# B&R Automation Studio project TD52 (part 74)

#### LX2.c
```c
/********************************************************************
 * COPYRIGHT -- Bernecker + Rainer Industrie-Elektronik Ges.m.b.H.
 ********************************************************************
 * Program: LX2
 * File: LX2.c
 * Author: 212566120
 * Created: Wed Apr 11 13:34:17 2018
 ********************************************************************
 * Implementation of program LX2
 ********************************************************************
 * Generated with B&R Automation Studio Target for Simulink V4.2
 * (ERT based)
 ********************************************************************/
#include "LX2.h"
#include "LX2_private.h"

/*  Defines */
#define LX2_POS_ZCSIG                  ((uint8_T)1U)
#define LX2_UNINITIALIZED_ZCSIG        ((uint8_T)3U)

/*  Data Types */

/**************************** GLOBAL DATA *************************************/
/*  Definitions */

/* Block signals (auto storage) */
struct BlockIO_LX2 LX2_B;

/* Block states (auto storage) */
struct D_Work_LX2 LX2_DWork;

/* Previous zero-crossings (trigger) states */
struct PrevZCSigStates_LX2 LX2_PrevZCSigState;

/* External inputs (root inport signals with auto storage) */
ExternalInputs_LX2 LX2_U;

/* External outputs (root outports fed by signals with auto storage) */
ExternalOutputs_LX2 LX2_Y;

/* Real-time model */
RT_MODEL_LX2 LX2_M_;
RT_MODEL_LX2 *const LX2_M = &LX2_M_;

/*  Declarations  */

/* Forward declaration for local functions */
static void LX2_my_split(real32_T x, real32_T *b_y1, real32_T *y2, struct fLX2* inst);
static void LX2_my_detect(real32_T x, real32_T *x1, real32_T *x2, struct fLX2* inst);
static real32_T LX2_my_split_i(real32_T x, struct fLX2* inst);
static void LX2_my_find(const real32_T V[11], real_T LowerLimit, real32_T
  UpperLimit, real_T p[11], struct fLX2* inst);
static void LX2_my_find_e(const real32_T V[11], real_T LowerLimit, real32_T
  UpperLimit, real_T p[11], struct fLX2* inst);
static void LX2_my_find_ex(const real32_T V[11], real32_T LowerLimit, real32_T
  UpperLimit, real_T p[11], struct fLX2* inst);
static void LX2_my_find_exl(const real32_T V[11], real32_T LowerLimit, real32_T
  UpperLimit, real_T p[11], struct fLX2* inst);
static void LX2_my_find_exlq(const real32_T V[11], real32_T LowerLimit, real_T
  UpperLimit, real_T p[11], struct fLX2* inst);
static void LX2_my_find_exlqw(const real32_T V[11], real32_T LowerLimit, real_T
  UpperLimit, real_T p[11], struct fLX2* inst);
static void LX2_my_find_exlqwy(const real32_T V[11], real_T p[11], struct fLX2* inst);
static real32_T LX2_sum(const real32_T x[11], struct fLX2* inst);
static void LX2_my_smoothing(const real32_T Pl[2], real32_T Pm[2], const
  real32_T Pr[2], real32_T slope_max, struct fLX2* inst);
static void LX2_interp1(const real32_T varargin_1[3], const real32_T varargin_2
  [3], const real32_T varargin_3[11], real32_T yi[11], struct fLX2* inst);
static void LX2_interp1_o(const real32_T varargin_1[4], const real32_T
  varargin_2[4], const real32_T varargin_3[11], real32_T yi[11], struct fLX2* inst);
static void LX2_interp1_o5pn4ly1(const real32_T varargin_1[11], const real32_T
  varargin_2[11], const real32_T varargin_3[11], real32_T yi[11], struct fLX2* inst);
static void LX2_interp1_o5(const real32_T varargin_1[5], const real32_T
  varargin_2[5], const real32_T varargin_3[11], real32_T yi[11], struct fLX2* inst);
static void LX2_interp1_o5p(const real32_T varargin_1[6], const real32_T
  varargin_2[6], const real32_T varargin_3[11], real32_T yi[11], struct fLX2* inst);
static void LX2_interp1_o5pn(const real32_T varargin_1[7], const real32_T
  varargin_2[7], const real32_T varargin_3[11], real32_T yi[11], struct fLX2* inst);
static real32_T LX2_interp1_o5pn4ly1e(const real32_T varargin_1[2], const
  real32_T varargin_2[2], real32_T varargin_3, struct fLX2* inst);
static void LX2_interp1_o5pn4(const real32_T varargin_1[8], const real32_T
  varargin_2[8], const real32_T varargin_3[11], real32_T yi[11], struct fLX2* inst);
static void LX2_interp1_o5pn4l(const real32_T varargin_1[9], const real32_T
  varargin_2[9], const real32_T varargin_3[11], real32_T yi[11], struct fLX2* inst);
static void LX2_interp1_o5pn4ly(const real32_T varargin_1[10], const real32_T
  varargin_2[10], const real32_T varargin_3[11], real32_T yi[11], struct fLX2* inst);
static void LX2_rdivide(const real32_T x[4], real_T y, real32_T z[4], struct fLX2* inst);

/* Forward declaration for local functions */
static void LX2_my_BPOC_enable_h(const real32_T splitfactor[4], boolean_T
  bLX2_enable, const real32_T rThreshold_save2map[2], boolean_T
  bExt_BPOC_learning_Stop, boolean_T bBPOC_enable[4], boolean_T
  bSave_BPOC_enable[4], struct fLX2* inst);
static void LX2_my_BPOC_enable(const real32_T splitfactor[4], boolean_T
  bLX2_enable, const real32_T rThreshold_save2map[2], boolean_T
  bExt_BPOC_learning_Stop, boolean_T bBPOC_enable[4], boolean_T
  bSave_BPOC_enable[4], struct fLX2* inst);
static void LX2_my_gasmixing(uint16_T iIdx_Gtyp_Dem, real32_T rGT_QualMix_1_2,
  real32_T rGT_RatioMix, boolean_T bLX2_enable, const real32_T
  rThreshold_save2map[2], boolean_T bExt_BPOC_learning_Stop, real32_T
  splitfactor_Gas[4], boolean_T bBPOC_enable[4], boolean_T bSave_BPOC_enable[4], struct fLX2* inst);

/***************************** FILE SCOPE DATA ********************************/

/*************************** FUNCTIONS ****************************************/

/* Lookup Binary Search Utility BINARYSEARCH_real32_T */
void BINARYSEARCH_real32_T(uint32_T *piLeft, uint32_T *piRght, real32_T u, const
  real32_T *pData, uint32_T iHi, struct fLX2* inst)
{
  /* Find the location of current input value in the data table. */
  *piLeft = 0U;
  *piRght = iHi;
  if (u <= pData[0] ) {
    /* Less than or equal to the smallest point in the table. */
    *piRght = 0U;
  } else if (u >= pData[iHi] ) {
    /* Greater than or equal to the largest point in the table. */
    *piLeft = iHi;
  } else {
    uint32_T i;

    /* Do a binary search. */
    while (( *piRght - *piLeft ) > 1U ) {
      /* Get the average of the left and right indices using to Floor rounding. */
      i = (*piLeft + *piRght) >> 1;

      /* Move either the right index or the left index so that */
      /*  LeftDataPoint <= CurrentValue < RightDataPoint */
      if (u < pData[i] ) {
        *piRght = i;
      } else {
        *piLeft = i;
      }
    }
  }
}

/* Lookup Utility LookUp_real32_T_real32_T */
void LookUp_real32_T_real32_T(real32_T *pY, const real32_T *pYData, real32_T u,
  const real32_T *pUData, uint32_T iHi, struct fLX2* inst)
{
  uint32_T iLeft;
  uint32_T iRght;
  BINARYSEARCH_real32_T( &(iLeft), &(iRght), u, pUData, iHi, inst);

  {
    real32_T lambda;
    if (pUData[iRght] > pUData[iLeft] ) {
      real32_T num;
      real32_T den;
      den = pUData[iRght];
      den = den - pUData[iLeft];
      num = u;
      num = num - pUData[iLeft];
      lambda = num / den;
    } else {
      lambda = 0.0F;
    }

    {
      real32_T yLeftCast;
      real32_T yRghtCast;
      yLeftCast = pYData[iLeft];
      yRghtCast = pYData[iRght];
      yLeftCast += lambda * ( yRghtCast - yLeftCast );
      (*pY) = yLeftCast;
    }
  }
}

real32_T rt_roundf(real32_T u, struct fLX2* inst)
{
  real32_T y;
  if ((real32_T)fabs(u) < 8.388608E+6F) {
    if (u >= 0.5F) {
      y = (real32_T)floor(u + 0.5F);
    } else if (u > -0.5F) {
      y = 0.0F;
    } else {
      y = (real32_T)ceil(u - 0.5F);
    }
  } else {
    y = u;
  }

  return y;
}

/* Function for MATLAB Function: '<S10>/Boost Pressure Offset Curve' */
static void LX2_my_split(real32_T x, real32_T *b_y1, real32_T *y2, struct fLX2* inst)
{
  real32_T t;

  /*  End od 'my_detect-function' */
  /*  ---------------------------------------------------------------------------------- */
  /* % my_split function */
  /* ************************************************************************** */
  /*  divides new measurement value up to neighborhood node points via leverage function */
  /*  */
  /*  Input:    x   ... Engine Power [%] */
  /*  Output:   y1  ... weighting of node left from x [-] */
  /*                  y2  ... weighting of node right from x [-] */
  /* ************************************************************************** */
  t = rt_roundf(x / 10.0F, inst) * 10.0F;

  /*  temporary var for decision and find neighborhood point */
  if (x < t) {
    /*  slope between the two neighboring points is positive */
    t -= x;
    *y2 = 1.0F - t / 10.0F;

    /*  weighting of node right from x */
    *b_y1 = 1.0F - (1.0F - t / 10.0F);

    /*  weighting of node left from x */
  } else if (x > t) {
    /*  slope between the two neighboring points is negative */
    t = x - t;
    *b_y1 = 1.0F - t / 10.0F;

    /*  weighting of node left from x */
    *y2 = 1.0F - (1.0F - t / 10.0F);

    /*  weighting of node right from x */
  } else if ((x == t) && (x != 100.0F)) {
    /*  x is exactly on node point; weighting factor is 1 */
    *b_y1 = 1.0F;
    *y2 = 0.0F;
  } else {
    /*  x is 100 */
    *b_y1 = 0.0F;
    *y2 = 1.0F;
  }
}

/* Function for MATLAB Function: '<S10>/Boost Pressure Offset Curve' */
static void LX2_my_detect(real32_T x, real32_T *x1, real32_T *x2, struct fLX2* inst)
{
  /*  End od 'BPOC.m' */
  /*  ---------------------------------------------------------------------------------- */
  /* % my_detect function */
  /* ************************************************************************** */
  /*  returns indices of affected node points due to new measurement value */
  /*  */
  /*  Input:    x   ... Engine Power [%] */
  /*  Output:   x1  ... index of left neighbouring node point [-] */
  /*                  x2  ... index of right neighbouring node point [-] */
  /* ************************************************************************** */
  if (!(x - (real32_T)floor(x / 2.0F) * 2.0F != 0.0F)) {
    /*  if x is exaclty on node -> manipulate x value with a super small value so that it is not lying on node anymore ;-) */
    x += 0.001F;
  }

  if (x <= 0.0F) {
    /*  input is limited to positive values  */
    *x1 = 1.0F;
    *x2 = 2.0F;
  } else if (x >= 100.0F) {
    /*  input is limited to values smaller than 100 (full load) */
    *x1 = 10.0F;
    *x2 = 11.0F;
  } else {
    *x1 = (real32_T)ceil(x / 10.0F);
    *x2 = *x1 + 1.0F;
  }
}

/* Function for MATLAB Function: '<S10>/Boost Pressure Offset Curve' */
static real32_T LX2_my_split_i(real32_T x, struct fLX2* inst)
{
  real32_T b_y1;
  real32_T t;

  /*  End od 'my_detect-function' */
  /*  ---------------------------------------------------------------------------------- */
  /* % my_split function */
  /* ************************************************************************** */
  /*  divides new measurement value up to neighborhood node points via leverage function */
  /*  */
  /*  Input:    x   ... Engine Power [%] */
  /*  Output:   y1  ... weighting of node left from x [-] */
  /*                  y2  ... weighting of node right from x [-] */
  /* ************************************************************************** */
  t = rt_roundf(x / 10.0F, inst) * 10.0F;

  /*  temporary var for decision and find neighborhood point */
  if (x < t) {
    /*  slope between the two neighboring points is positive */
    /*  weighting of node right from x */
    b_y1 = 1.0F - (1.0F - (t - x) / 10.0F);

    /*  weighting of node left from x */
  } else if (x > t) {
    /*  slope between the two neighboring points is negative */
    b_y1 = 1.0F - (x - t) / 10.0F;

    /*  weighting of node left from x */
    /*  weighting of node right from x */
  } else if ((x == t) && (x != 100.0F)) {
    /*  x is exactly on node point; weighting factor is 1 */
    b_y1 = 1.0F;
  } else {
    /*  x is 100 */
    b_y1 = 0.0F;
  }

  return b_y1;
}

/* Function for MATLAB Function: '<S10>/Boost Pressure Offset Curve' */
static void LX2_my_find(const real32_T V[11], real_T LowerLimit, real32_T
  UpperLimit, real_T p[11], struct fLX2* inst)
{
  real32_T i;
  int32_T b_i;
  int32_T b;
  int32_T i_0;

  /*  end of 'my_smoothing-function' */
  /* ---------------------------------------------------------------------------------- */
  /* % my_find */
  /* ************************************************************************** */
  /*  returns indices of already measured points depending on 'mode' and 'Limits' */
  /*  */
  /*  Input:    V                   ... binary map (vector, 11 elements, boolean) */
  /*                LowerLimit   ... lower search boundary (scalar) */
  /*                UpperLimit   ... upper search boundary (scalar) */
  /*                mode            ... 'first' -> returns first 2 indices */
  /*                                      ... 'last' -> returns last 2 indices */
  /*                                      ... 'all' -> returns all found indices */
  /*  */
  /*  Output: Pm	...	middle point of triangle  (vector, 2 elements, Pm(1)->[%], Pm(2)->[mbar]) */
  /* ************************************************************************** */
  for (i_0 = 0; i_0 < 11; i_0++) {
    p[i_0] = 0.0;
  }

  /*  fixed allocated vector for saving indices */
  /*  -> function will return indices of first two elements which were found */
  /*  -> always write 2 values to p - no need for more, thats why 2=hard coded */
  i_0 = 0;
  b = (int32_T)((1.0F - (real32_T)LowerLimit) + UpperLimit);
  for (b_i = 0; b_i < b; b_i++) {
    i = (real32_T)LowerLimit + (real32_T)b_i;
    if ((V[(int32_T)i - 1] != 0.0F) && (i_0 < 2)) {
      p[i_0] = i;
      i_0++;
    }
  }

  /*  -> function will return indices of last two elements which were found        */
  /*  -> always write 2 values to p - no need for more, thats why 2=hard coded   */
  /*  end 'if-function' */
  /*  end of 'my_find-function'  */
  /* ---------------------------------------------------------------------------------- */
}

/* Function for MATLAB Function: '<S10>/Boost Pressure Offset Curve' */
static void LX2_my_find_e(const real32_T V[11], real_T LowerLimit, real32_T
  UpperLimit, real_T p[11], struct fLX2* inst)
{
  real32_T i;
  int32_T b_i;
  int32_T b;
  int32_T i_0;

  /*  end of 'my_smoothing-function' */
  /* ---------------------------------------------------------------------------------- */
  /* % my_find */
  /* ************************************************************************** */
  /*  returns indices of already measured points depending on 'mode' and 'Limits' */
  /*  */
  /*  Input:    V                   ... binary map (vector, 11 elements, boolean) */
  /*                LowerLimit   ... lower search boundary (scalar) */
  /*                UpperLimit   ... upper search boundary (scalar) */
  /*                mode            ... 'first' -> returns first 2 indices */
  /*                                      ... 'last' -> returns last 2 indices */
  /*                                      ... 'all' -> returns all found indices */
  /*  */
  /*  Output: Pm	...	middle point of triangle  (vector, 2 elements, Pm(1)->[%], Pm(2)->[mbar]) */
  /* ************************************************************************** */
  for (i_0 = 0; i_0 < 11; i_0++) {
    p[i_0] = 0.0;
  }

  /*  fixed allocated vector for saving indices */
  /*  -> function will return indices of first two elements which were found */
  /*  -> always write 2 values to p - no need for more, thats why 2=hard coded */
  i_0 = 2;
  b = (int32_T)-((-1.0F - UpperLimit) + (real32_T)LowerLimit);
  for (b_i = 0; b_i < b; b_i++) {
    i = UpperLimit + -(real32_T)b_i;
    if ((V[(int32_T)i - 1] != 0.0F) && (i_0 > 0)) {
      p[i_0 - 1] = i;
      i_0--;
    }
  }

  /*  -> function will return all indices which were found - used for smoothing-function and interpolation of all points */
  /*  -> loop writes values into p from end to start of vector - smoothing-function need this order */
  /*  end 'if-function' */
  /*  end of 'my_find-function'  */
  /* ---------------------------------------------------------------------------------- */
}

/* Function for MATLAB Function: '<S10>/Boost Pressure Offset Curve' */
static void LX2_my_find_ex(const real32_T V[11], real32_T LowerLimit, real32_T
  UpperLimit, real_T p[11], struct fLX2* inst)
{
  real32_T i;
  int32_T b_i;
  int32_T b;
  int32_T i_0;

  /*  end of 'my_smoothing-function' */
  /* ---------------------------------------------------------------------------------- */
  /* % my_find */
  /* ************************************************************************** */
  /*  returns indices of already measured points depending on 'mode' and 'Limits' */
  /*  */
  /*  Input:    V                   ... binary map (vector, 11 elements, boolean) */
  /*                LowerLimit   ... lower search boundary (scalar) */
  /*                UpperLimit   ... upper search boundary (scalar) */
  /*                mode            ... 'first' -> returns first 2 indices */
  /*                                      ... 'last' -> returns last 2 indices */
  /*                                      ... 'all' -> returns all found indices */
  /*  */
  /*  Output: Pm	...	middle point of triangle  (vector, 2 elements, Pm(1)->[%], Pm(2)->[mbar]) */
  /* ************************************************************************** */
  for (i_0 = 0; i_0 < 11; i_0++) {
    p[i_0] = 0.0;
  }

  /*  fixed allocated vector for saving indices */
  /*  -> function will return indices of first two elements which were found */
  /*  -> always write 2 values to p - no need for more, thats why 2=hard coded */
  i_0 = 0;
  b = (int32_T)((1.0F - LowerLimit) + UpperLimit);
  for (b_i = 0; b_i < b; b_i++) {
    i = LowerLimit + (real32_T)b_i;
    if ((V[(int32_T)i - 1] != 0.0F) && (i_0 < 2)) {
      p[i_0] = i;
      i_0++;
    }
  }

  /*  -> function will return indices of last two elements which were found        */
  /*  -> always write 2 values to p - no need for more, thats why 2=hard coded   */
  /*  end 'if-function' */
  /*  end of 'my_find-function'  */
  /* ---------------------------------------------------------------------------------- */
}

/* Function for MATLAB Function: '<S10>/Boost Pressure Offset Curve' */
static void LX2_my_find_exl(const real32_T V[11], real32_T LowerLimit, real32_T
  UpperLimit, real_T p[11], struct fLX2* inst)
{
  real32_T i;
  int32_T b_i;
  int32_T b;
  int32_T i_0;

  /*  end of 'my_smoothing-function' */
  /* ---------------------------------------------------------------------------------- */
  /* % my_find */
  /* ************************************************************************** */
  /*  returns indices of already measured points depending on 'mode' and 'Limits' */
  /*  */
  /*  Input:    V                   ... binary map (vector, 11 elements, boolean) */
  /*                LowerLimit   ... lower search boundary (scalar) */
  /*                UpperLimit   ... upper search boundary (scalar) */
  /*                mode            ... 'first' -> returns first 2 indices */
  /*                                      ... 'last' -> returns last 2 indices */
  /*                                      ... 'all' -> returns all found indices */
  /*  */
  /*  Output: Pm	...	middle point of triangle  (vector, 2 elements, Pm(1)->[%], Pm(2)->[mbar]) */
  /* ************************************************************************** */
  for (i_0 = 0; i_0 < 11; i_0++) {
    p[i_0] = 0.0;
  }

  /*  fixed allocated vector for saving indices */
  /*  -> function will return indices of first two elements which were found */
  /*  -> always write 2 values to p - no need for more, thats why 2=hard coded */
  i_0 = 2;
  b = (int32_T)-((-1.0F - UpperLimit) + LowerLimit);
  for (b_i = 0; b_i < b; b_i++) {
    i = UpperLimit + -(real32_T)b_i;
    if ((V[(int32_T)i - 1] != 0.0F) && (i_0 > 0)) {
      p[i_0 - 1] = i;
      i_0--;
    }
  }

  /*  -> function will return all indices which were found - used for smoothing-function and interpolation of all points */
  /*  -> loop writes values into p from end to start of vector - smoothing-function need this order */
  /*  end 'if-function' */
  /*  end of 'my_find-function'  */
  /* ---------------------------------------------------------------------------------- */
}

/* Function for MATLAB Function: '<S10>/Boost Pressure Offset Curve' */
static void LX2_my_find_exlq(const real32_T V[11], real32_T LowerLimit, real_T
  UpperLimit, real_T p[11], struct fLX2* inst)
{
  real32_T i;
  int32_T b_i;
  int32_T b;
  int32_T i_0;

  /*  end of 'my_smoothing-function' */
  /* ---------------------------------------------------------------------------------- */
  /* % my_find */
  /* ************************************************************************** */
  /*  returns indices of already measured points depending on 'mode' and 'Limits' */
  /*  */
  /*  Input:    V                   ... binary map (vector, 11 elements, boolean) */
  /*                LowerLimit   ... lower search boundary (scalar) */
  /*                UpperLimit   ... upper search boundary (scalar) */
  /*                mode            ... 'first' -> returns first 2 indices */
  /*                                      ... 'last' -> returns last 2 indices */
  /*                                      ... 'all' -> returns all found indices */
  /*  */
  /*  Output: Pm	...	middle point of triangle  (vector, 2 elements, Pm(1)->[%], Pm(2)->[mbar]) */
  /* ************************************************************************** */
  for (i_0 = 0; i_0 < 11; i_0++) {
    p[i_0] = 0.0;
  }

  /*  fixed allocated vector for saving indices */
  /*  -> function will return indices of first two elements which were found */
  /*  -> always write 2 values to p - no need for more, thats why 2=hard coded */
  i_0 = 0;
  b = (int32_T)((1.0F - LowerLimit) + (real32_T)UpperLimit);
  for (b_i = 0; b_i < b; b_i++) {
    i = LowerLimit + (real32_T)b_i;
    if ((V[(int32_T)i - 1] != 0.0F) && (i_0 < 2)) {
      p[i_0] = i;
      i_0++;
    }
  }

  /*  -> function will return indices of last two elements which were found        */
  /*  -> always write 2 values to p - no need for more, thats why 2=hard coded   */
  /*  end 'if-function' */
  /*  end of 'my_find-function'  */
  /* ---------------------------------------------------------------------------------- */
}

/* Function for MATLAB Function: '<S10>/Boost Pressure Offset Curve' */
static void LX2_my_find_exlqw(const real32_T V[11], real32_T LowerLimit, real_T
  UpperLimit, real_T p[11], struct fLX2* inst)
{
  real32_T i;
  int32_T b_i;
  int32_T b;
  int32_T i_0;

  /*  end of 'my_smoothing-function' */
  /* ---------------------------------------------------------------------------------- */
  /* % my_find */
  /* ************************************************************************** */
  /*  returns indices of already measured points depending on 'mode' and 'Limits' */
  /*  */
  /*  Input:    V                   ... binary map (vector, 11 elements, boolean) */
  /*                LowerLimit   ... lower search boundary (scalar) */
  /*                UpperLimit   ... upper search boundary (scalar) */
  /*                mode            ... 'first' -> returns first 2 indices */
  /*                                      ... 'last' -> returns last 2 indices */
  /*                                      ... 'all' -> returns all found indices */
  /*  */
  /*  Output: Pm	...	middle point of triangle  (vector, 2 elements, Pm(1)->[%], Pm(2)->[mbar]) */
  /* ************************************************************************** */
  for (i_0 = 0; i_0 < 11; i_0++) {
    p[i_0] = 0.0;
  }

  /*  fixed allocated vector for saving indices */
  /*  -> function will return indices of first two elements which were found */
  /*  -> always write 2 values to p - no need for more, thats why 2=hard coded */
  i_0 = 2;
  b = (int32_T)-((-1.0F - (real32_T)UpperLimit) + LowerLimit);
  for (b_i = 0; b_i < b; b_i++) {
    i = (real32_T)UpperLimit + -(real32_T)b_i;
    if ((V[(int32_T)i - 1] != 0.0F) && (i_0 > 0)) {
      p[i_0 - 1] = i;
      i_0--;
    }
  }

  /*  -> function will return all indices which were found - used for smoothing-function and interpolation of all points */
  /*  -> loop writes values into p from end to start of vector - smoothing-function need this order */
  /*  end 'if-function' */
  /*  end of 'my_find-function'  */
  /* ---------------------------------------------------------------------------------- */
}

/* Function for MATLAB Function: '<S10>/Boost Pressure Offset Curve' */
static void LX2_my_find_exlqwy(const real32_T V[11], real_T p[11], struct fLX2* inst)
{
  real_T j;
  int32_T i;

  /*  end of 'my_smoothing-function' */
  /* ---------------------------------------------------------------------------------- */
  /* % my_find */
  /* ************************************************************************** */
  /*  returns indices of already measured points depending on 'mode' and 'Limits' */
  /*  */
  /*  Input:    V                   ... binary map (vector, 11 elements, boolean) */
  /*                LowerLimit   ... lower search boundary (scalar) */
  /*                UpperLimit   ... upper search boundary (scalar) */
  /*                mode            ... 'first' -> returns first 2 indices */
  /*                                      ... 'last' -> returns last 2 indices */
  /*                                      ... 'all' -> returns all found indices */
  /*  */
  /*  Output: Pm	...	middle point of triangle  (vector, 2 elements, Pm(1)->[%], Pm(2)->[mbar]) */
  /* ************************************************************************** */
  for (i = 0; i < 11; i++) {
    p[i] = 0.0;
  }

  /*  fixed allocated vector for saving indices */
  /*  -> function will return indices of first two elements which were found */
  /*  -> always write 2 values to p - no need for more, thats why 2=hard coded */
  j = 11.0;
  for (i = 0; i < 11; i++) {
    if (V[10 - i] != 0.0F) {
      p[(int32_T)j - 1] = 11.0 + -(real_T)i;
      j--;
    }
  }

  /*  end 'if-function' */
  /*  end of 'my_find-function'  */
  /* ---------------------------------------------------------------------------------- */
}

/* Function for MATLAB Function: '<S10>/Boost Pressure Offset Curve' */
static real32_T LX2_sum(const real32_T x[11], struct fLX2* inst)
{
  real32_T y;
  int32_T k;
  y = x[0];
  for (k = 0; k < 10; k++) {
    y += x[k + 1];
  }

  return y;
}

/* Function for MATLAB Function: '<S10>/Boost Pressure Offset Curve' */
static void LX2_my_smoothing(const real32_T Pl[2], real32_T Pm[2], const
  real32_T Pr[2], real32_T slope_max, struct fLX2* inst)
{
  real32_T Pmr_max;
  real32_T Pmr_min;
  real32_T Pml_max;
  real32_T Pml_min;

  /*  End of 'my_split-function' */
  /* ---------------------------------------------------------------------------------- */
  /* % my_smoothing function */
  /* ************************************************************************** */
  /*  returns new delta_p2s at Pm, if one of the slopes of the triangel is */
  /*  greater than slope_max */
  /*  */
  /*  Input:    Pl      ... left point of triangle (vector, 2 elements, Pl(1)->[%], Pl(2)->[mbar]) */
  /*                Pm    ... middle point of triangle  (vector, 2 elements, Pm(1)->[%], Pm(2)->[mbar]) */
  /*                Pr      ... right point of triangle (vector, 2 elements, Pr(1)->[%], Pr(2)->[mbar]) */
  /*                slope_max   ... max. slope within triangle [mbar/%-Engine Power] */
  /*  */
  /*  Output: Pm	...	middle point of triangle  (vector, 2 elements, Pm(1)->[%], Pm(2)->[mbar]) */
  /* ************************************************************************** */
  /*  calc slope right */
  /*  calc slope left */
  if (((real32_T)fabs((Pr[1] - Pm[1]) / (Pr[0] - Pm[0])) > slope_max) ||
      ((real32_T)fabs((Pm[1] - Pl[1]) / (Pm[0] - Pl[0])) > slope_max)) {
    /*  one of the slopes are not within the limit */
    Pmr_max = (Pr[0] - Pm[0]) * slope_max + Pr[1];

    /*  max. allowed value for Pm depending on Pr */
    Pmr_min = Pr[1] - (Pr[0] - Pm[0]) * slope_max;

    /*  min. value allowed for Pm depending on Pr */
    Pml_max = (Pm[0] - Pl[0]) * slope_max + Pl[1];

    /*  max. value allowed for Pm depending on Pl */
    Pml_min = Pl[1] - (Pm[0] - Pl[0]) * slope_max;

    /*  min. value allowed for Pm depending on Pl */
    /*  make Pm to Pm_new   */
    if ((Pmr_max >= Pml_max) && (Pmr_min <= Pml_min) && (Pr[0] - Pm[0] > Pm[0] -
         Pl[0])) {
      /*  bigger right area contains left area */
      if (Pm[1] >= Pml_max) {
        Pm[1] = Pml_max;
      } else {
        if (Pm[1] <= Pml_min) {
          Pm[1] = Pml_min;
        }
      }
    } else if ((Pml_max >= Pmr_max) && (Pml_min <= Pmr_min) && (Pm[0] - Pl[0] >
                Pr[0] - Pm[0])) {
      /*  bigger left area contains right area */
      if (Pm[1] >= Pmr_max) {
        Pm[1] = Pmr_max;
      } else {
        if (Pm[1] <= Pmr_min) {
          Pm[1] = Pmr_min;
        }
      }
    } else if ((Pmr_max <= Pml_max) && (Pmr_max >= Pml_min)) {
      /*  required slope can be reached by changing Pm to the closest value in the overlap area */
      if (Pm[1] >= Pmr_max) {
        Pm[1] = Pmr_max;
      } else {
        if (Pm[1] <= Pml_min) {
          Pm[1] = Pml_min;
        }
      }
    } else if ((Pmr_min >= Pml_min) && (Pmr_min <= Pml_max)) {
      /*  required slope can be reached by changing Pm to the closest value in the overlap area */
      if (Pm[1] >= Pml_max) {
        Pm[1] = Pml_max;
      } else {
        if (Pm[1] <= Pmr_min) {
          Pm[1] = Pmr_min;
        }
      }
    } else if (Pmr_max < Pml_min) {
      /*  required slope cannot be reached by changing Pm in pos. direction -> right slope of triange is set to slope_max */
      Pm[1] = Pmr_max;
    } else {
      if (Pmr_min > Pml_max) {
        /*  required slope cannot be reached by changing Pm in neg. direction -> right slope of triange is set to slope_max */
        Pm[1] = Pmr_min;
      }
    }

    /*  make Pm_new to Pm */
  }

  /*  end smoothing-algorithm */
  /*  if slopes are okay, delta_p2s @ Pm will not be changed -> Pm-Input == Pm-Output */
}

/* Function for MATLAB Function: '<S10>/Boost Pressure Offset Curve' */
static void LX2_interp1(const real32_T varargin_1[3], const real32_T varargin_2
  [3], const real32_T varargin_3[11], real32_T yi[11], struct fLX2* inst)
{
  real32_T y[3];
  real32_T x[3];
  real32_T r;
  int32_T low_i;
  int32_T low_ip;
  int32_T high_i;
  int32_T i;
  y[0] = varargin_2[0];
  y[1] = varargin_2[1];
  y[2] = varargin_2[2];
  x[0] = varargin_1[0];
  x[1] = varargin_1[1];
  x[2] = varargin_1[2];
  for (i = 0; i < 11; i++) {
    yi[i] = 0.0F;
  }

  if (varargin_1[1] < varargin_1[0]) {
    x[0] = varargin_1[2];
    x[2] = varargin_1[0];
    y[0] = varargin_2[2];
    y[2] = varargin_2[0];
  }

  for (i = 0; i < 11; i++) {
    if (!((varargin_3[i] > x[2]) || (varargin_3[i] < x[0]))) {
      low_i = 0;
      low_ip = 2;
      high_i = 3;
      while (high_i > low_ip) {
        if (varargin_3[i] >= varargin_1[1]) {
          low_i = 1;
          low_ip = 3;
        } else {
          high_i = 2;
        }
      }

      r = (varargin_3[i] - x[low_i]) / (x[low_i + 1] - x[low_i]);
      if (y[low_i + 1] == y[low_i]) {
        yi[i] = y[low_i];
      } else {
        yi[i] = (1.0F - r) * y[low_i] + y[low_i + 1] * r;
      }
    }
  }
}

/* Function for MATLAB Function: '<S10>/Boost Pressure Offset Curve' */
static void LX2_interp1_o(const real32_T varargin_1[4], const real32_T
  varargin_2[4], const real32_T varargin_3[11], real32_T yi[11], struct fLX2* inst)
{
  real32_T y[4];
  real32_T x[4];
  real32_T r;
  int32_T low_i;
  int32_T low_ip;
  int32_T high_i;
  int32_T mid_i;
  int32_T i;
  y[0] = varargin_2[0];
  y[1] = varargin_2[1];
  y[2] = varargin_2[2];
  y[3] = varargin_2[3];
  x[0] = varargin_1[0];
  x[1] = varargin_1[1];
  x[2] = varargin_1[2];
  x[3] = varargin_1[3];
  for (i = 0; i < 11; i++) {
    yi[i] = 0.0F;
  }

  if (varargin_1[1] < varargin_1[0]) {
    x[0] = varargin_1[3];
    x[3] = varargin_1[0];
    x[1] = varargin_1[2];
    x[2] = varargin_1[1];
    y[0] = varargin_2[3];
    y[3] = varargin_2[0];
    y[1] = varargin_2[2];
    y[2] = varargin_2[1];
  }

  for (i = 0; i < 11; i++) {
    if (!((varargin_3[i] > x[3]) || (varargin_3[i] < x[0]))) {
      low_i = 1;
      low_ip = 2;
      high_i = 4;
      while (high_i > low_ip) {
        mid_i = (low_i + high_i) >> 1;
        if (varargin_3[i] >= x[mid_i - 1]) {
          low_i = mid_i;
          low_ip = mid_i + 1;
        } else {
          high_i = mid_i;
        }
      }

      r = (varargin_3[i] - x[low_i - 1]) / (x[low_i] - x[low_i - 1]);
      if (y[low_i - 1] == y[low_i]) {
        yi[i] = y[low_i - 1];
      } else {
        yi[i] = (1.0F - r) * y[low_i - 1] + r * y[low_i];
      }
    }
  }
}

/* Function for MATLAB Function: '<S10>/Boost Pressure Offset Curve' */
static void LX2_interp1_o5pn4ly1(const real32_T varargin_1[11], const real32_T
  varargin_2[11], const real32_T varargin_3[11], real32_T yi[11], struct fLX2* inst)
{
  real32_T y[11];
  real32_T x[11];
  real32_T r;
  int32_T ixright;
  int32_T low_ip;
  int32_T high_i;
  int32_T mid_i;
  int32_T i;
  for (i = 0; i < 11; i++) {
    y[i] = varargin_2[i];
    x[i] = varargin_1[i];
    yi[i] = 0.0F;
  }

  if (varargin_1[1] < varargin_1[0]) {
    for (i = 0; i < 5; i++) {
      r = x[i];
      x[i] = x[10 - i];
      x[10 - i] = r;
    }

    i = 0;
    for (ixright = 10; i + 1 < ixright + 1; ixright--) {
      r = y[i];
      y[i] = y[ixright];
      y[ixright] = r;
      i++;
    }
  }

  for (i = 0; i < 11; i++) {
    if (!((varargin_3[i] > x[10]) || (varargin_3[i] < x[0]))) {
      ixright = 1;
      low_ip = 2;
      high_i = 11;
      while (high_i > low_ip) {
        mid_i = (ixright + high_i) >> 1;
        if (varargin_3[i] >= x[mid_i - 1]) {
          ixright = mid_i;
          low_ip = mid_i + 1;
        } else {
          high_i = mid_i;
        }
      }

      if (ixright != 0) {
        r = (varargin_3[i] - x[ixright - 1]) / (x[ixright] - x[ixright - 1]);
        if (y[ixright - 1] == y[ixright]) {
          yi[i] = y[ixright - 1];
        } else {
          yi[i] = (1.0F - r) * y[ixright - 1] + r * y[ixright];
        }
      }
    }
  }
}

/* Function for MATLAB Function: '<S10>/Boost Pressure Offset Curve' */
static void LX2_interp1_o5(const real32_T varargin_1[5], const real32_T
  varargin_2[5], const real32_T varargin_3[11], real32_T yi[11], struct fLX2* inst)
{
  real32_T y[5];
  real32_T x[5];
  real32_T r;
  int32_T low_i;
  int32_T low_ip;
  int32_T high_i;
  int32_T mid_i;
  int32_T i;
  for (i = 0; i < 5; i++) {
    y[i] = varargin_2[i];
    x[i] = varargin_1[i];
  }

  for (i = 0; i < 11; i++) {
    yi[i] = 0.0F;
  }

  if (varargin_1[1] < varargin_1[0]) {
    r = x[0];
    x[0] = x[4];
    x[4] = r;
    r = x[1];
    x[1] = x[3];
    x[3] = r;
    r = y[0];
    y[0] = y[4];
    y[4] = r;
    r = y[1];
    y[1] = y[3];
    y[3] = r;
  }

  for (i = 0; i < 11; i++) {
    if (!((varargin_3[i] > x[4]) || (varargin_3[i] < x[0]))) {
      low_i = 1;
      low_ip = 2;
      high_i = 5;
      while (high_i > low_ip) {
        mid_i = (low_i + high_i) >> 1;
        if (varargin_3[i] >= x[mid_i - 1]) {
          low_i = mid_i;
          low_ip = mid_i + 1;
        } else {
          high_i = mid_i;
        }
      }

      r = (varargin_3[i] - x[low_i - 1]) / (x[low_i] - x[low_i - 1]);
      if (y[low_i - 1] == y[low_i]) {
        yi[i] = y[low_i - 1];
      } else {
        yi[i] = (1.0F - r) * y[low_i - 1] + r * y[low_i];
      }
    }
  }
}

/* Function for MATLAB Function: '<S10>/Boost Pressure Offset Curve' */
static void LX2_interp1_o5p(const real32_T varargin_1[6], const real32_T
  varargin_2[6], const real32_T varargin_3[11], real32_T yi[11], struct fLX2* inst)
{
  real32_T y[6];
  real32_T x[6];
  real32_T r;
  int32_T low_i;
  int32_T low_ip;
  int32_T high_i;
  int32_T mid_i;
  int32_T i;
  for (i = 0; i < 6; i++) {
    y[i] = varargin_2[i];
    x[i] = varargin_1[i];
  }

  for (i = 0; i < 11; i++) {
    yi[i] = 0.0F;
  }

  if (varargin_1[1] < varargin_1[0]) {
    r = x[0];
    x[0] = x[5];
    x[5] = r;
    r = x[1];
    x[1] = x[4];
    x[4] = r;
    r = x[2];
    x[2] = x[3];
    x[3] = r;
    r = y[0];
    y[0] = y[5];
    y[5] = r;
    r = y[1];
    y[1] = y[4];
    y[4] = r;
    r = y[2];
    y[2] = y[3];
    y[3] = r;
  }

  for (i = 0; i < 11; i++) {
    if (!((varargin_3[i] > x[5]) || (varargin_3[i] < x[0]))) {
      low_i = 1;
      low_ip = 2;
      high_i = 6;
      while (high_i > low_ip) {
        mid_i = (low_i + high_i) >> 1;
        if (varargin_3[i] >= x[mid_i - 1]) {
          low_i = mid_i;
          low_ip = mid_i + 1;
        } else {
          high_i = mid_i;
        }
      }

      if (low_i != 0) {
        r = (varargin_3[i] - x[low_i - 1]) / (x[low_i] - x[low_i - 1]);
        if (y[low_i - 1] == y[low_i]) {
          yi[i] = y[low_i - 1];
        } else {
          yi[i] = (1.0F - r) * y[low_i - 1] + r * y[low_i];
        }
      }
    }
  }
}

/* Function for MATLAB Function: '<S10>/Boost Pressure Offset Curve' */
static void LX2_interp1_o5pn(const real32_T varargin_1[7], const real32_T
  varargin_2[7], const real32_T varargin_3[11], real32_T yi[11], struct fLX2* inst)
{
  real32_T y[7];
  real32_T x[7];
  real32_T r;
  int32_T low_i;
  int32_T low_ip;
  int32_T high_i;
  int32_T mid_i;
  int32_T i;
  for (i = 0; i < 7; i++) {
    y[i] = varargin_2[i];
    x[i] = varargin_1[i];
  }

  for (i = 0; i < 11; i++) {
    yi[i] = 0.0F;
  }

  if (varargin_1[1] < varargin_1[0]) {
    r = x[0];
    x[0] = x[6];
    x[6] = r;
    r = x[1];
    x[1] = x[5];
    x[5] = r;
    r = x[2];
    x[2] = x[4];
    x[4] = r;
    r = y[0];
    y[0] = y[6];
    y[6] = r;
    r = y[1];
    y[1] = y[5];
    y[5] = r;
    r = y[2];
    y[2] = y[4];
    y[4] = r;
  }

  for (i = 0; i < 11; i++) {
    if (!((varargin_3[i] > x[6]) || (varargin_3[i] < x[0]))) {
      low_i = 1;
      low_ip = 2;
      high_i = 7;
      while (high_i > low_ip) {
        mid_i = (low_i + high_i) >> 1;
        if (varargin_3[i] >= x[mid_i - 1]) {
          low_i = mid_i;
          low_ip = mid_i + 1;
        } else {
          high_i = mid_i;
        }
      }

      r = (varargin_3[i] - x[low_i - 1]) / (x[low_i] - x[low_i - 1]);
      if (y[low_i - 1] == y[low_i]) {
        yi[i] = y[low_i - 1];
      } else {
        yi[i] = (1.0F - r) * y[low_i - 1] + r * y[low_i];
      }
    }
  }
}

/* Function for MATLAB Function: '<S10>/Boost Pressure Offset Curve' */
static real32_T LX2_interp1_o5pn4ly1e(const real32_T varargin_1[2], const
  real32_T varargin_2[2], real32_T varargin_3, struct fLX2* inst)
{
  real32_T yi;
  real32_T r;
  int32_T ixleft;
  int32_T ixright;
  real32_T y_idx;
  real32_T x_idx;
  real32_T x_idx_0;
  real32_T y_idx_0;
  y_idx_0 = varargin_2[0];
  y_idx = varargin_2[1];
  x_idx = varargin_1[0];
  x_idx_0 = varargin_1[1];
  yi = 0.0F;
  if (varargin_1[1] < varargin_1[0]) {
    x_idx = varargin_1[1];
    x_idx_0 = varargin_1[0];
    ixleft = 1;
    ixright = 2;
    while (ixleft < ixright) {
      r = y_idx_0;
      y_idx_0 = y_idx;
      y_idx = r;
      ixleft = 2;
      ixright = 1;
    }
  }

  if (!((varargin_3 > x_idx_0) || (varargin_3 < x_idx))) {
    r = (varargin_3 - x_idx) / (x_idx_0 - x_idx);
    if (y_idx_0 == y_idx) {
      yi = y_idx_0;
    } else {
      yi = (1.0F - r) * y_idx_0 + r * y_idx;
    }
  }

  return yi;
}

/* Function for MATLAB Function: '<S10>/Boost Pressure Offset Curve' */
static void LX2_interp1_o5pn4(const real32_T varargin_1[8], const real32_T
  varargin_2[8], const real32_T varargin_3[11], real32_T yi[11], struct fLX2* inst)
{
  real32_T y[8];
  real32_T x[8];
  real32_T r;
  int32_T low_i;
  int32_T low_ip;
  int32_T high_i;
  int32_T mid_i;
  int32_T i;
  for (i = 0; i < 8; i++) {
    y[i] = varargin_2[i];
    x[i] = varargin_1[i];
  }

  for (i = 0; i < 11; i++) {
    yi[i] = 0.0F;
  }

  if (varargin_1[1] < varargin_1[0]) {
    r = x[0];
    x[0] = x[7];
    x[7] = r;
    r = x[1];
    x[1] = x[6];
    x[6] = r;
    r = x[2];
    x[2] = x[5];
    x[5] = r;
    r = x[3];
    x[3] = x[4];
    x[4] = r;
    r = y[0];
    y[0] = y[7];
    y[7] = r;
    r = y[1];
    y[1] = y[6];
    y[6] = r;
    r = y[2];
    y[2] = y[5];
    y[5] = r;
    r = y[3];
    y[3] = y[4];
    y[4] = r;
  }

  for (i = 0; i < 11; i++) {
    if (!((varargin_3[i] > x[7]) || (varargin_3[i] < x[0]))) {
      low_i = 1;
      low_ip = 2;
      high_i = 8;
      while (high_i > low_ip) {
        mid_i = (low_i + high_i) >> 1;
        if (varargin_3[i] >= x[mid_i - 1]) {
          low_i = mid_i;
          low_ip = mid_i + 1;
        } else {
          high_i = mid_i;
        }
      }

      r = (varargin_3[i] - x[low_i - 1]) / (x[low_i] - x[low_i - 1]);
      if (y[low_i - 1] == y[low_i]) {
        yi[i] = y[low_i - 1];
      } else {
        yi[i] = (1.0F - r) * y[low_i - 1] + r * y[low_i];
      }
    }
  }
}

/* Function for MATLAB Function: '<S10>/Boost Pressure Offset Curve' */
static void LX2_interp1_o5pn4l(const real32_T varargin_1[9], const real32_T
  varargin_2[9], const real32_T varargin_3[11], real32_T yi[11], struct fLX2* inst)
{
  real32_T y[9];
  real32_T x[9];
  real32_T r;
  int32_T low_i;
  int32_T low_ip;
  int32_T high_i;
  int32_T mid_i;
  int32_T i;
  for (i = 0; i < 9; i++) {
    y[i] = varargin_2[i];
    x[i] = varargin_1[i];
  }

  for (i = 0; i < 11; i++) {
    yi[i] = 0.0F;
  }

  if (varargin_1[1] < varargin_1[0]) {
    r = x[0];
    x[0] = x[8];
    x[8] = r;
    r = x[1];
    x[1] = x[7];
    x[7] = r;
    r = x[2];
    x[2] = x[6];
    x[6] = r;
    r = x[3];
    x[3] = x[5];
    x[5] = r;
    r = y[0];
    y[0] = y[8];
    y[8] = r;
    r = y[1];
    y[1] = y[7];
    y[7] = r;
    r = y[2];
    y[2] = y[6];
    y[6] = r;
    r = y[3];
    y[3] = y[5];
    y[5] = r;
  }

  for (i = 0; i < 11; i++) {
    if (!((varargin_3[i] > x[8]) || (varargin_3[i] < x[0]))) {
      low_i = 1;
      low_ip = 2;
      high_i = 9;
      while (high_i > low_ip) {
        mid_i = (low_i + high_i) >> 1;
        if (varargin_3[i] >= x[mid_i - 1]) {
          low_i = mid_i;
          low_ip = mid_i + 1;
        } else {
          high_i = mid_i;
        }
      }

      r = (varargin_3[i] - x[low_i - 1]) / (x[low_i] - x[low_i - 1]);
      if (y[low_i - 1] == y[low_i]) {
        yi[i] = y[low_i - 1];
      } else {
        yi[i] = (1.0F - r) * y[low_i - 1] + r * y[low_i];
      }
    }
  }
}

/* Function for MATLAB Function: '<S10>/Boost Pressure Offset Curve' */
static void LX2_interp1_o5pn4ly(const real32_T varargin_1[10], const real32_T
  varargin_2[10], const real32_T varargin_3[11], real32_T yi[11], struct fLX2* inst)
{
  real32_T y[10];
  real32_T x[10];
  real32_T r;
  int32_T low_i;
  int32_T low_ip;
  int32_T high_i;
  int32_T mid_i;
  int32_T i;
  for (i = 0; i < 10; i++) {
    y[i] = varargin_2[i];
    x[i] = varargin_1[i];
  }

  for (i = 0; i < 11; i++) {
    yi[i] = 0.0F;
  }

  if (varargin_1[1] < varargin_1[0]) {
    for (i = 0; i < 5; i++) {
      r = x[i];
      x[i] = x[9 - i];
      x[9 - i] = r;
    }

    for (i = 0; i < 5; i++) {
      r = y[i];
      y[i] = y[9 - i];
      y[9 - i] = r;
    }
  }

  for (i = 0; i < 11; i++) {
    if (!((varargin_3[i] > x[9]) || (varargin_3[i] < x[0]))) {
      low_i = 1;
      low_ip = 2;
      high_i = 10;
      while (high_i > low_ip) {
        mid_i = (low_i + high_i) >> 1;
        if (varargin_3[i] >= x[mid_i - 1]) {
          low_i = mid_i;
          low_ip = mid_i + 1;
        } else {
          high_i = mid_i;
        }
      }

      if (low_i != 0) {
        r = (varargin_3[i] - x[low_i - 1]) / (x[low_i] - x[low_i - 1]);
        if (y[low_i - 1] == y[low_i]) {
          yi[i] = y[low_i - 1];
        } else {
          yi[i] = (1.0F - r) * y[low_i - 1] + r * y[low_i];
        }
      }
    }
  }
}

/* Function for MATLAB Function: '<S10>/Boost Pressure Offset Curve' */
static void LX2_rdivide(const real32_T x[4], real_T y, real32_T z[4], struct fLX2* inst)
{
  z[0] = x[0] / (real32_T)y;
  z[1] = x[1] / (real32_T)y;
  z[2] = x[2] / (real32_T)y;
  z[3] = x[3] / (real32_T)y;
}

/*
 * Output and update for atomic system:
 *    '<S10>/Boost Pressure Offset Curve'
 *    '<S11>/Boost Pressure Offset Curve'
 *    '<S12>/Boost Pressure Offset Curve'
 *    '<S13>/Boost Pressure Offset Curve'
 */
void LX2_BoostPressureOffsetCurve(real32_T rtu_x, real32_T rtu_y, const real32_T
  rtu_IN_offset[11], const boolean_T rtu_IN_measured[11], const real32_T
  rtu_LPs[3], boolean_T rtu_Lp_c_ena, real32_T rtu_s_max, real32_T rtu_s_maxEx,
  uint16_T rtu_w1, uint16_T rtu_w2, uint16_T rtu_w3, uint16_T rtu_w4, real32_T
  rtu_limit_value, boolean_T rtu_Enable, rtB_BoostPressureOffsetCurve_LX *localB, struct fLX2* inst)
{
  real32_T x;
  real32_T y;
  boolean_T Lp_c_ena;
  real32_T s_max;
  real32_T s_maxEx;
  real32_T DBUG_sInt;
  real32_T DBUG_sExt_right;
  real32_T DBUG_sExt_left;
  real32_T P_LPs[11];
  real32_T P[44];
  real32_T P_new[44];
  real32_T slope;
  real32_T delta_slope;
  real_T p[11];
  real32_T aa;
  real32_T aa_0;
  real32_T b;
  real32_T b_0;
  real32_T w;
  real32_T w_0;
  real32_T w_1;
  real32_T f[2];
  boolean_T guard = FALSE;
  int32_T i;
  real32_T tmp[4];
  real32_T tmp_0[2];
  real32_T P_new_0[2];
  real32_T P_new_1[11];
  real32_T P_new_2[11];
  real32_T P_new_3[10];
  real32_T P_new_4[10];
  real32_T P_new_5[9];
  real32_T P_new_6[9];
  real32_T P_new_7[8];
  real32_T P_new_8[8];
  real32_T P_new_9[7];
  real32_T P_new_a[7];
  real32_T P_new_b[6];
  real32_T P_new_c[6];
  real32_T P_new_d[5];
  real32_T P_new_e[5];
  real32_T P_new_f[4];
  real32_T P_new_g[4];
  real32_T P_new_h[3];
  real32_T P_new_i[3];
  real32_T P_new_j[2];
  real32_T P_new_k[2];
  real32_T Lp_idx;
  real32_T Lp_idx_0;

  /* MATLAB Function 'Boost Pressure Offset Map/Boost Pressure Offset Curve': '<S15>:1' */
  x = rtu_x;
  y = rtu_y;
  Lp_c_ena = rtu_Lp_c_ena;
  s_max = rtu_s_max;
  s_maxEx = rtu_s_maxEx;

  /* % Header */
  /*  This Function manipulates the Boost-Pressure-Offset-Curve (BPOC) */
  /*  depending on a new delta_p2s @ %-EnginePower */
  /*  Rev 1 : Christian Schneider, 24.08.2018 */
  /*  Rev 1.1 : Enrico Maran, 18.01.2021    //extrapolation at 0% load limited to 10% of control limit   */
  /*  Rev 2.0 : Enrico Maran, 22.06.2021    //integrated Leanox point at low load */
  /*  Input:    x                   ...   normiert Engine Power [%],[0...100], (scalar) */
  /*                y                   ...   delta_p2s [bar], (scalar) */
  /*                IN_offset      ...   delta_p2s [bar] @ node points, (vector, 11 elements, scalar) */
  /*                IN_measured ... binary map of already measured points [-], (vector, 11 elements, boolean) */
  /*                LPs               ...   position of Leanox points (half/full load/low load), [%-Engine Power] (vector, 3 elements, scalar) */
  /*                Lp_c_ena         ...   Leanox point c enabled (~25% load) [-], (boolean) */
  /*                s_max           ...   max. allowed slope of BPOC (interpolation) [bar/%-Engine Power], (scalar) */
  /*                s_maxEx       ...   max. allowed slope of BPOC towards Leanox-Points (extrapolation)  [bar/%-Engine Power], (scalar) */
  /*                w1                ...   weighting factor for Leanox Point 1 (0% load), [-], (integer) */
  /*                w2                ...   weighting factor for Leanox Point 2 (~50% load, able to vary), [-], (integer) */
  /*                w3                ...   weighting factor for Leanox Point 3 (100% load), [-], (integer) */
  /*                w4                ...   weighting factor for Leanox Point c (~25% load), [-], (integer) */
  /*                limit_value       ...   BPOC limit value [bar], (scalar) */
  /*                Enable         ...   enable function [-], (boolean) */
  /*  */
  /*  Output: OUT_offset      ...   delta p2s [bar] @ node points, (vector, 11 elements, scalar) */
  /*                OUT_measured ... binary map of already measured points [-], (vector, 11 elements, boolean) */
  /*                Nodes             ... Nodes of BPOC [%-Engine Power], (vector, 11 elements, scalar) */
  /*                e                      ... error between new delta_p2s value and interpolated BPOC-value [bar], (scalar) */
  /*  */
  /*  Debug-Outbuts: DBUG_a     ...     nodes of BPOC which are affected by new measurement value [-], (vector, 2 elements, scalar) -> DBUG_a(1)=left node, DBUG_a(1)=right node */
  /*                              DBUG_b     ...     weighting of affected node points due to leverage function [-], (vector, 2 elements, scalar) -> DBUG_b(1)=left node, DBUG_b(1)=right node */
  /*                              DBUG_Lp   ...     location of leanox points on map (indices) [-], (vector, 3 elements, scalar) -> DBUG_Lp(1)=leanox point @ 0kW, DBUG_Lp(2)=leanox point @ ~50 load, DBUG_Lp(3)=leanox point @ 100 load, DBUG_Lp(4)=leanox point @ ~25 load */
  /*                              DBUG_s     ...     s ... calculated slopes (Interpolation/Extrapolation), [vector, 3 elements, scalar]-> DBUG_sInt ... slope between affected nodes, DBUG_sExt_left ... extrapolation slope to the left side, DBUG_sExt_right ... extrapolation slope to the left side */
  /* % Main Function BPOC */
  /*  node points of BPOC <<| LX2_FunReq-4 |>> */
  /*  Initzialisation of DBUG variables */
  /*  set DBUG_sInt to -1 -> only for debugging */
  DBUG_sExt_right = -1.0F;

  /*  set DBUG_sExt_right to -1 -> only for debugging */
  DBUG_sExt_left = -1.0F;

  /*  set DBUG_sExt_left to -1 -> only for debugging */
  if (rtu_Enable) {
    /*  enable manipulation of BPOC */
    /* % check input parameter and creating P-Matrix */
    /*  x-Parameter -> normiert Engine Power [%] */
    /*  (only values between "0 <= x <= 100" are allowed) */
    if (rtu_x < 0.0F) {
      x = 0.0F;
    } else {
      if (rtu_x > 100.0F) {
        x = 100.0F;
      }
    }

    /* --------------------------------------------- */
    /*  s_max & s_maxEx -> slope limit between two nodes (interpolation/extrapolation) [bar/%-EngPower] */
    /*  (only values between "0 <= s_max <= 3" are allowed) */
    if (rtu_s_max < 0.0F) {
      s_max = 0.0F;
    } else {
      if (rtu_s_max > 10.0F) {
        s_max = 3.0F;
      }
    }

    if (rtu_s_maxEx < 0.0F) {
      s_maxEx = 0.0F;
    } else {
      if (rtu_s_maxEx > s_max) {
        /*  s_maxEx is not allowed to be greater than s_max */
        s_maxEx = s_max;
      }
    }

    /* --------------------------------------------- */
    /*  w1, w2, w3 -> weighting factors for teached in leanox points [-] */
    /*  (only values between "0 <= s_max <= 10" are allowed) */
    /*  casting is needed because further calculations are not possible with datatype integer */
    w_1 = (real32_T)rtu_w4;

    /* --------------------------------------------- */
    /*  Creating P-Matrix (11-by-4 Matrix) */
    /*  */
    /*  Column 1, P(:,1) -> Node points */
    /*  Column 2, P(:,2) -> delta_p2s offset values */
    /*  Column 3, P(:,3) -> binary map of already measured points */
    /*  Column 4, P(:,4) -> binary map of Leanox points */
    /*  */
    /*  Example: */
    /*     0        0           0       1 */
    /*    10        0.01356     0       0 */
    /*    20        0.01476     0       0 */
    /*    30        0.02952     0       0 */
    /*    40        0.04428     0       1 */
    /*    50        0.04430     1       0 */
    /*    60        0.04432     0       0 */
    /*    70        0.04434     0       0 */
    /*    80        0.04436     1       0 */
    /*    90        0.04438     1       0 */
    /*   100        0.04440     1       1 */
    /*  *********************************************************************** */
    /*  Handling of Leanox Points  */
    /*        -> all Leanox Points are lying direct on a node point  */
    /*        -> if teached in Leanox point is not lying direct on node point - it will be moved to the most closest one */
    /*        -> weighting factor of leanox point will be weighted again depending on distance of real/teached leanox point */
    /*  *********************************************************************** */
    for (i = 0; i < 11; i++) {
      P_LPs[i] = 0.0F;
    }

    /*  create 4th column of P-Matrix */
    Lp_idx = 0.0F;

    /*  vector for saving indices of Leanox points depending on Node points */
    /*  Leanox Point 1 at 0% load (fix) */
    P_LPs[0] = 1.0F;

    /*  Lp1 always at node 1 -> 0% load */
    /*  Lp1 always at node 1 -> 0% load => Index 1 */
    /* ********************************* */
    /*  Leanox Point 2 at half load (variable -> depending on location of teached in point) */
    LX2_my_split(rtu_LPs[0], &slope, &delta_slope, inst);
    LX2_my_detect(rtu_LPs[0], &aa, &aa_0, inst);
    if (slope > delta_slope) {
      P_LPs[(int32_T)aa - 1] = 1.0F;
      w = (real32_T)rtu_w2 * slope;

      /*  weighting factor w2 of Lp2 will be weighted again depending on distance of real Leanox point */
      Lp_idx_0 = aa;

      /*  saving index of Leanox point 2 */
    } else {
      /*  bb1 < bb2 */
      P_LPs[(int32_T)aa_0 - 1] = 1.0F;
      w = (real32_T)rtu_w2 * delta_slope;

      /*  weighting factor w2 of Lp2 will be weighted again depending on distance of real Leanox point */
      Lp_idx_0 = aa_0;

      /*  saving index of Leanox point 2 */
    }

    /* ********************************* */
    /*  Leanox Point 3 at full load (fix) */
    P_LPs[10] = 1.0F;

    /*  Lp3 always at node 11 -> 100% load */
    /*  Lp3 always at node 11 -> 100% load => Index 11 */
    /* ********************************* */
    /*  adjustment of weighting factor due to position/distance of real Leanox point */
    if ((rtu_LPs[1] > 100.0F) && (rtu_LPs[1] < 110.0F)) {
      /*  Lp3 is between 100% and 110% load */
      w_0 = (1.0F - (rtu_LPs[1] - 100.0F) / 10.0F) * (real32_T)rtu_w3;
    } else if ((rtu_LPs[1] > 90.0F) && (rtu_LPs[1] <= 100.0F)) {
      /*  LP is between 90% and 100% load */
      w_0 = (1.0F - LX2_my_split_i(rtu_LPs[1], inst)) * (real32_T)rtu_w3;
    } else {
      w_0 = 0.0F;

      /*  LP not in defined range (>110% or <90%) */
    }

    /* ********************************* */
    /*  Leanox Point c at low load (~25%) (variable -> depending on location of teached in point) */
    if (rtu_Lp_c_ena) {
      if ((rtu_LPs[2] < rtu_LPs[0]) && (rtu_LPs[2] >= 10.0F)) {
        /*  if actual load reference of 25% Leanox point is lower than 50% Leanox point and >=10% load */
        LX2_my_split(rtu_LPs[2], &slope, &delta_slope, inst);
        LX2_my_detect(rtu_LPs[2], &aa, &aa_0, inst);
        if (slope > delta_slope) {
          P_LPs[(int32_T)aa - 1] = 1.0F;
          w_1 = (real32_T)rtu_w4 * slope;

          /*  weighting factor w4 of Lp_c will be weighted again depending on distance of real Leanox point */
          Lp_idx = aa;

          /*  saving index of Leanox point c */
        } else {
          /*  bb1_Lp_c < bb2_Lp_c */
          P_LPs[(int32_T)aa_0 - 1] = 1.0F;
          w_1 = (real32_T)rtu_w4 * delta_slope;

          /*  weighting factor w4 of Lp_c will be weighted again depending on distance of real Leanox point */
          Lp_idx = aa_0;

          /*  saving index of Leanox point c */
        }
      } else {
        /*  assign to 25% leanox point same values as 50% point */
        w_1 = w;
        Lp_idx = Lp_idx_0;
      }
    }

    /* ********************************* */
    /*  casting is needed because P-Matrix is not able to contain different datatypes */
    for (i = 0; i < 11; i++) {
      P[i] = 10.0F * (real32_T)i;
    }

    for (i = 0; i < 11; i++) {
      P[i + 11] = rtu_IN_offset[i];
    }

    for (i = 0; i < 11; i++) {
      P[i + 22] = (real32_T)rtu_IN_measured[i];
    }

    for (i = 0; i < 11; i++) {
      P[i + 33] = P_LPs[i];
    }

    /*  crating P-matrix */
    /* ---------------------------------------------------------------------------------- */
    /* % Detection of new Measurement point + Split via Leverage Function */
    for (i = 0; i < 44; i++) {
      P_new[i] = P[i];
    }

    /*  make old matrix to new matrix */
    /*  detects which nodes of BPOC are affected by new measurement value <<| LX2_FunReq-17 |>> */
    LX2_my_detect(x, &aa, &aa_0, inst);

    /*  divides new measurement value up to neighborhood node points via leverage function <<| LX2_FunReq-17 |>> */
    LX2_my_split(x, &b, &b_0, inst);

    /* ---------------------------------------------------------------------------------- */
    /* % Handling of measured values    */
    /*  <<| LX2_FunReq-17 |>><<| LX2_FunReq-18 |>><<| LX2_FunReq-15 |>> */
    P_new[(int32_T)aa + 10] = ((P[(int32_T)aa + 10] * (1.0F - b) + rtu_y * b) +
      P[(int32_T)aa + 10]) / 2.0F;

    /*  old and new value are weighted depending on split-function */
    P_new[(int32_T)aa + 21] = 1.0F;

    /*  writing 1 to the binary map -> already measured point */
    P_new[(int32_T)aa_0 + 10] = ((P[(int32_T)aa_0 + 10] * (1.0F - b_0) + rtu_y *
      b_0) + P[(int32_T)aa_0 + 10]) / 2.0F;

    /*  old and new value are weighted depending on split-function */
    P_new[(int32_T)aa_0 + 21] = 1.0F;

    /*  writing 1 to the binary map -> already measured point */
    slope = (P_new[(int32_T)aa_0 + 10] - P_new[(int32_T)aa + 10]) / (P_new
      [(int32_T)aa_0 - 1] - P_new[(int32_T)aa - 1]);
    DBUG_sInt = slope;

    /*  map calculated slope to DBUG_sInt variable */
    if ((real32_T)fabs(slope) > s_max) {
      /*  check if slope is within limit */
      delta_slope = (real32_T)fabs(slope) - s_max;

      /*  calc delta between max. allowed slope and actual slope */
      if (slope > 0.0F) {
        /*  slope is positive */
        P_new[(int32_T)aa + 10] += (P_new[(int32_T)aa_0 - 1] - P_new[(int32_T)aa
          - 1]) * (delta_slope * b_0);

        /*  move left point up (pos.), depending on delta_slope */
        P_new[(int32_T)aa_0 + 10] -= (P_new[(int32_T)aa_0 - 1] - P_new[(int32_T)
          aa - 1]) * (delta_slope * b);

        /*  move right point down (neg.), dependting on delta_slope */
      } else {
        if (slope < 0.0F) {
          /*  slope is negative */
          P_new[(int32_T)aa + 10] -= (P_new[(int32_T)aa_0 - 1] - P_new[(int32_T)
            aa - 1]) * (delta_slope * b_0);

          /*  move left point down (neg.), depending on delta_slope */
          P_new[(int32_T)aa_0 + 10] += (P_new[(int32_T)aa_0 - 1] - P_new
            [(int32_T)aa - 1]) * (delta_slope * b);

          /*  move right point up (pos.), depending on delta_slope */
        }
      }
    }

    /* ---------------------------------------------------------------------------------- */
    /* % manipulation of teached LEANOX Points */
    /*  <<| LX2_FunReq-14 |>> */
    /*  Leanox point 1 - Lp1 %%%%%%%%%%%%%%%%%%%%%%%%%%%%%%%%%%%%%% */
    if (x < P[(int32_T)Lp_idx_0 - 1]) {
      if (!(rtu_Lp_c_ena && (Lp_idx < Lp_idx_0))) {
        /*  x lies between  Lp1 and Lp2  */
        LX2_my_find(*(real32_T (*)[11])&P_new[22], 1.0, Lp_idx_0, p, inst);

        /*  indices of  two most closest node points with already measured values -> right side of Lp1 */
        slope = (P_new[(int32_T)p[1] + 10] - P_new[(int32_T)p[0] + 10]) /
          (P_new[(int32_T)p[1] - 1] - P_new[(int32_T)p[0] - 1]);

        /*  calc slope between points, which were found before */
        DBUG_sExt_left = slope;

        /*  map calculated slope to DBUG_sExt_left variable */
        if ((real32_T)fabs(slope) > s_maxEx) {
          /*  check if slope okay, otherwise limit it to s_maxEx */
          if (slope < 0.0F) {
            slope = -s_maxEx;
          } else {
            slope = s_maxEx;
          }
        }

        P_new[11] = ((P_new[(int32_T)p[0] + 10] - (P_new[(int32_T)p[0] - 1] -
          P_new[0]) * slope) + (real32_T)rtu_w1 * P[11]) / (1.0F + (real32_T)
          rtu_w1);

        /*  Extrapolation to Lp1 */
        if (P_new[22] == 0.0F) {
          /*  if LP1 is not measured apply additional limitation to extrapolated value */
          slope = rtu_limit_value * 0.1F;
          if (P_new[11] <= slope) {
            slope = P_new[11];
          }

          delta_slope = -rtu_limit_value * 0.1F;
          if (delta_slope >= slope) {
            P_new[11] = delta_slope;
          } else {
            P_new[11] = slope;
          }

          /*  limitation to 10% of control range */
        }
      } else {
        guard = TRUE;
      }
    } else {
      guard = TRUE;
    }

    if (guard && ((x < P[(int32_T)Lp_idx - 1]) && rtu_Lp_c_ena && (Lp_idx <
          Lp_idx_0))) {
      /*  x lies between  Lp1 and Lp_c     */
      LX2_my_find(*(real32_T (*)[11])&P_new[22], 1.0, Lp_idx, p, inst);

      /*  indices of  two most closest node points with already measured values -> right side of Lp1 */
      slope = (P_new[(int32_T)p[1] + 10] - P_new[(int32_T)p[0] + 10]) / (P_new
        [(int32_T)p[1] - 1] - P_new[(int32_T)p[0] - 1]);

      /*  calc slope between points, which were found before */
      DBUG_sExt_left = slope;

      /*  map calculated slope to DBUG_sExt_left variable */
      if ((real32_T)fabs(slope) > s_maxEx) {
        /*  check if slope okay, otherwise limit it to s_maxEx */
        if (slope < 0.0F) {
          slope = -s_maxEx;
        } else {
          slope = s_maxEx;
        }
      }

      P_new[11] = ((P_new[(int32_T)p[0] + 10] - (P_new[(int32_T)p[0] - 1] -
        P_new[0]) * slope) + (real32_T)rtu_w1 * P[11]) / (1.0F + (real32_T)
        rtu_w1);

      /*  Extrapolation to Lp1 */
      if (P_new[22] == 0.0F) {
        /*  if LP1 is not measured apply additional limitation to extrapolated value */
        slope = rtu_limit_value * 0.1F;
        if (P_new[11] <= slope) {
          slope = P_new[11];
        }

        delta_slope = -rtu_limit_value * 0.1F;
        if (delta_slope >= slope) {
          P_new[11] = delta_slope;
        } else {
          P_new[11] = slope;
        }

        /*  limitation to 10% of control range */
      }
    }

    /* ---------------------------------------------------------------------------------- */
    /*  <<| LX2_FunReq-14 |>> */
    /*  Leanox point c (~25% load) - Lp4  %%%%%%%%%%%%%%%%%%%%%%%%%%%%%%%%%%%%%% */
    if (rtu_Lp_c_ena && (Lp_idx < Lp_idx_0)) {
      /*  apply only if Lp_c is enabled, otherwise consider standard 3 Leanox point logic  */
      if (x < P[(int32_T)Lp_idx - 1]) {
        /*  x lies between  Lp1 and Lp_c  */
        LX2_my_find_e(*(real32_T (*)[11])&P_new[22], 1.0, Lp_idx, p, inst);

        /*  indices of  two most closest node points with already measured values -> left side of Lp_c */
        /*  new Measurment point is between two nodes */
        slope = (P_new[(int32_T)p[1] + 10] - P_new[(int32_T)p[0] + 10]) /
          (P_new[(int32_T)p[1] - 1] - P_new[(int32_T)p[0] - 1]);

        /*  calc slope between points, which were found before */
        DBUG_sExt_right = slope;

        /*  map calculated slope to DBUG_sExt_right variable */
        if ((real32_T)fabs(slope) > s_maxEx) {
          /*  check if slope okay, otherwise limit it to s_maxEx */
          if (slope < 0.0F) {
            slope = -s_maxEx;
          } else {
            slope = s_maxEx;
          }
        }

        P_new[(int32_T)Lp_idx + 10] = (((P_new[(int32_T)Lp_idx - 1] - P_new
          [(int32_T)p[1] - 1]) * slope + P_new[(int32_T)p[1] + 10]) + P[(int32_T)
          Lp_idx + 10] * w_1) / (1.0F + w_1);

        /*  Extrapolation to Lp2 */
      } else if ((x > P[(int32_T)Lp_idx - 1]) && (x < P[(int32_T)Lp_idx_0 - 1]))
      {
        /*  x lies between  Lp_c and Lp2  */
        LX2_my_find_ex(*(real32_T (*)[11])&P_new[22], Lp_idx, Lp_idx_0, p, inst);

        /*  indices of  two most closest node points with already measured values -> right side of Lp_c */
        slope = (P_new[(int32_T)p[1] + 10] - P_new[(int32_T)p[0] + 10]) /
          (P_new[(int32_T)p[1] - 1] - P_new[(int32_T)p[0] - 1]);

        /*  calc slope between points, which were found before */
        DBUG_sExt_left = slope;

        /*  map calculated slope to DBUG_sExt_left variable */
        if ((real32_T)fabs(slope) > s_maxEx) {
          /*  check if slope okay, otherwise limit it to s_maxEx */
          if (slope < 0.0F) {
            slope = -s_maxEx;
          } else {
            slope = s_maxEx;
          }
        }

        P_new[(int32_T)Lp_idx + 10] = ((P_new[(int32_T)p[0] + 10] - (P_new
          [(int32_T)p[0] - 1] - P_new[(int32_T)Lp_idx - 1]) * slope) + P
          [(int32_T)Lp_idx + 10] * w_1) / (1.0F + w_1);
      } else {
        if (P[(int32_T)Lp_idx - 1] == x) {
          P_new[(int32_T)Lp_idx + 10] = (P[(int32_T)Lp_idx + 10] * w_1 + P_new
            [(int32_T)Lp_idx + 10]) / (1.0F + w_1);

          /*  measurement point lies exactly on node of Lp_c */
        }
      }
    }

    /* ---------------------------------------------------------------------------------- */
    /*  <<| LX2_FunReq-14 |>> */
    /*  Leanox point 2 - Lp2 %%%%%%%%%%%%%%%%%%%%%%%%%%%%%%%%%%%%%% */
    guard = FALSE;
    if (x < P[(int32_T)Lp_idx_0 - 1]) {
      if (!(rtu_Lp_c_ena && (Lp_idx < Lp_idx_0))) {
        /*  x lies between  Lp1 and Lp2  */
        LX2_my_find_e(*(real32_T (*)[11])&P_new[22], 1.0, Lp_idx_0, p, inst);

        /*  indices of  two most closest node points with already measured values -> left side of Lp2 */
        /*  new Measurment point is between two nodes */
        slope = (P_new[(int32_T)p[1] + 10] - P_new[(int32_T)p[0] + 10]) /
          (P_new[(int32_T)p[1] - 1] - P_new[(int32_T)p[0] - 1]);

        /*  calc slope between points, which were found before */
        DBUG_sExt_right = slope;

        /*  map calculated slope to DBUG_sExt_right variable */
        if ((real32_T)fabs(slope) > s_maxEx) {
          /*  check if slope okay, otherwise limit it to s_maxEx */
          if (slope < 0.0F) {
            slope = -s_maxEx;
          } else {
            slope = s_maxEx;
          }
        }

        P_new[(int32_T)Lp_idx_0 + 10] = (((P_new[(int32_T)Lp_idx_0 - 1] - P_new
          [(int32_T)p[1] - 1]) * slope + P_new[(int32_T)p[1] + 10]) + P[(int32_T)
          Lp_idx_0 + 10] * w) / (1.0F + w);

        /*  Extrapolation to Lp2 */
      } else {
        guard = TRUE;
      }
    } else {
      guard = TRUE;
    }

    if (guard) {
      if ((x < P[(int32_T)Lp_idx_0 - 1]) && (x > P[(int32_T)Lp_idx - 1]) &&
          rtu_Lp_c_ena && (Lp_idx < Lp_idx_0)) {
        /*  x lies between  Lp_c and Lp2  */
        LX2_my_find_exl(*(real32_T (*)[11])&P_new[22], Lp_idx, Lp_idx_0, p, inst);

        /*  indices of  two most closest node points with already measured values -> left side of Lp2 */
        /*  new Measurment point is between two nodes */
        slope = (P_new[(int32_T)p[1] + 10] - P_new[(int32_T)p[0] + 10]) /
          (P_new[(int32_T)p[1] - 1] - P_new[(int32_T)p[0] - 1]);

        /*  calc slope between points, which were found before */
        DBUG_sExt_right = slope;

        /*  map calculated slope to DBUG_sExt_right variable */
        if ((real32_T)fabs(slope) > s_maxEx) {
          /*  check if slope okay, otherwise limit it to s_maxEx */
          if (slope < 0.0F) {
            slope = -s_maxEx;
          } else {
            slope = s_maxEx;
          }
        }

        P_new[(int32_T)Lp_idx_0 + 10] = (((P_new[(int32_T)Lp_idx_0 - 1] - P_new
          [(int32_T)p[1] - 1]) * slope + P_new[(int32_T)p[1] + 10]) + P[(int32_T)
          Lp_idx_0 + 10] * w) / (1.0F + w);

        /*  Extrapolation to Lp2 */
      } else if (x > P[(int32_T)Lp_idx_0 - 1]) {
        /*  x lies between  Lp2 and Lp3  */
        LX2_my_find_exlq(*(real32_T (*)[11])&P_new[22], Lp_idx_0, 11.0, p, inst);

        /*  indices of  two most closest node points with already measured values -> right side of Lp2 */
        slope = (P_new[(int32_T)p[1] + 10] - P_new[(int32_T)p[0] + 10]) /
          (P_new[(int32_T)p[1] - 1] - P_new[(int32_T)p[0] - 1]);

        /*  calc slope between points, which were found before */
        DBUG_sExt_left = slope;

        /*  map calculated slope to DBUG_sExt_left variable */
        if ((real32_T)fabs(slope) > s_maxEx) {
          /*  check if slope okay, otherwise limit it to s_maxEx */
          if (slope < 0.0F) {
            slope = -s_maxEx;
          } else {
            slope = s_maxEx;
          }
        }

        P_new[(int32_T)Lp_idx_0 + 10] = ((P_new[(int32_T)p[0] + 10] - (P_new
          [(int32_T)p[0] - 1] - P_new[(int32_T)Lp_idx_0 - 1]) * slope) + P
          [(int32_T)Lp_idx_0 + 10] * w) / (1.0F + w);
      } else {
        if (P[(int32_T)Lp_idx_0 - 1] == x) {
          P_new[(int32_T)Lp_idx_0 + 10] = (P[(int32_T)Lp_idx_0 + 10] * w +
            P_new[(int32_T)Lp_idx_0 + 10]) / (1.0F + w);

          /*  measurement point lies exactly on node of Lp2 */
        }
      }
    }

    /* ---------------------------------------------------------------------------------- */
    /*  <<| LX2_FunReq-14 |>> */
    /*  Leanox point 3 - Lp3 %%%%%%%%%%%%%%%%%%%%%%%%%%%%%%%%%%%%%% */
    if (x > P[(int32_T)Lp_idx_0 - 1]) {
      /*  x lies between  Lp2 and Lp3  */
      LX2_my_find_exlqw(*(real32_T (*)[11])&P_new[22], Lp_idx_0, 11.0, p, inst);

      /*  indices of  two most closest node points with already measured values -> left side of Lp3 */
      slope = (P_new[(int32_T)p[1] + 10] - P_new[(int32_T)p[0] + 10]) / (P_new
        [(int32_T)p[1] - 1] - P_new[(int32_T)p[0] - 1]);

      /*  calc slope between points, which were found before */
      DBUG_sExt_right = slope;

      /*  map calculated slope to DBUG_sExt_right variable */
      if ((real32_T)fabs(slope) > s_maxEx) {
        /*  check if slope okay, otherwise limit it to s_maxEx */
        if (slope < 0.0F) {
          slope = -s_maxEx;
        } else {
          slope = s_maxEx;
        }
      }

      P_new[21] = (((P_new[10] - P_new[(int32_T)p[1] - 1]) * slope + P_new
                    [(int32_T)p[1] + 10]) + w_0 * P[21]) / (1.0F + w_0);
    }

    /* ---------------------------------------------------------------------------------- */
    /* % BPOC smoothening */
    /*  <<| LX2_FunReq-15 |>> to guarantee all slopes of BPOC are within the required limit  */
    for (i = 0; i < 11; i++) {
      P_LPs[i] = P_new[22 + i];
    }

    /*  binary map of node points with already measured values */
    P_LPs[0] = 1.0F;
    P_LPs[(int32_T)Lp_idx_0 - 1] = 1.0F;
    P_LPs[10] = 1.0F;

    /*  consider Leanox points in map */
    if (rtu_Lp_c_ena && (Lp_idx < Lp_idx_0)) {
      /*  consider also Leanox point c if relevant */
      P_LPs[(int32_T)Lp_idx - 1] = 1.0F;
    }

    LX2_my_find_exlqwy(P_LPs, p, inst);

    /*  find all indices of j, where already measured values available */
    /*  for-loop applies smoothing-function from biggest to smallest indices (from 100% load -> 0% load) */
    slope = LX2_sum(P_LPs, inst) - 3.0F;
    for (i = 0; i < (int32_T)(slope + 1.0F); i++) {
      /*  Input of my_smoothing: right point of triangle */
      /*  Input of my_smoothing: middle point of triangle */
      /*  Input of my_smoothing: left point of triangle */
      /*  call smoothening-function */
      f[0] = P_new[(int32_T)p[(int32_T)(10.0F - (real32_T)i) - 1] - 1];
      f[1] = P_new[(int32_T)p[(int32_T)(10.0F - (real32_T)i) - 1] + 10];
      P_new_j[0] = P_new[(int32_T)p[(int32_T)(9.0F - (real32_T)i) - 1] - 1];
      P_new_j[1] = P_new[(int32_T)p[(int32_T)(9.0F - (real32_T)i) - 1] + 10];
      P_new_k[0] = P_new[(int32_T)p[(int32_T)(11.0F - (real32_T)i) - 1] - 1];
      P_new_k[1] = P_new[(int32_T)p[(int32_T)(11.0F - (real32_T)i) - 1] + 10];
      LX2_my_smoothing(P_new_j, f, P_new_k, s_max, inst);
      P_new[(int32_T)p[(int32_T)(10.0F - (real32_T)i) - 1] + 10] = f[1];
    }

    /*  end smoothening */
    /* % Interpolation */
    /*  <<| LX2_FunReq-16 |>> */
    /*  interpolates complete BPOC depending on how many measured points are already available */
    for (i = 0; i < 11; i++) {
      P_LPs[i] = P_new[22 + i];
    }

    P_LPs[0] = 1.0F;
    P_LPs[(int32_T)Lp_idx_0 - 1] = 1.0F;
    P_LPs[10] = 1.0F;
    if (Lp_c_ena && (Lp_idx < Lp_idx_0)) {
      /*  consider also Leanox point c if relevant */
      P_LPs[(int32_T)Lp_idx - 1] = 1.0F;
    }

    LX2_my_find_exlqwy(P_LPs, p, inst);

    /*  find all indices for interpolation algorithm */
    if (LX2_sum(P_LPs, inst) == 3.0F) {
      P_new_h[0] = P_new[(int32_T)p[8] - 1];
      P_new_h[1] = P_new[(int32_T)p[9] - 1];
      P_new_h[2] = P_new[(int32_T)p[10] - 1];
      P_new_i[0] = P_new[(int32_T)p[0] + 10];
      P_new_i[1] = P_new[(int32_T)p[1] + 10];
      P_new_i[2] = P_new[(int32_T)p[2] + 10];
      for (i = 0; i < 11; i++) {
        P_LPs[i] = (*(real32_T (*)[11])&P_new[0])[i];
      }

      LX2_interp1(P_new_h, P_new_i, P_LPs, *(real32_T (*)[11])&P_new[11], inst);
    } else if (LX2_sum(P_LPs, inst) == 4.0F) {
      P_new_f[0] = P_new[(int32_T)p[7] - 1];
      P_new_f[1] = P_new[(int32_T)p[8] - 1];
      P_new_f[2] = P_new[(int32_T)p[9] - 1];
      P_new_f[3] = P_new[(int32_T)p[10] - 1];
      P_new_g[0] = P_new[(int32_T)p[7] + 10];
      P_new_g[1] = P_new[(int32_T)p[8] + 10];
      P_new_g[2] = P_new[(int32_T)p[9] + 10];
      P_new_g[3] = P_new[(int32_T)p[10] + 10];
      for (i = 0; i < 11; i++) {
        P_LPs[i] = (*(real32_T (*)[11])&P_new[0])[i];
      }

      LX2_interp1_o(P_new_f, P_new_g, P_LPs, *(real32_T (*)[11])&P_new[11], inst);
    } else if (LX2_sum(P_LPs, inst) == 5.0F) {
      P_new_d[0] = P_new[(int32_T)p[6] - 1];
      P_new_d[1] = P_new[(int32_T)p[7] - 1];
      P_new_d[2] = P_new[(int32_T)p[8] - 1];
      P_new_d[3] = P_new[(int32_T)p[9] - 1];
      P_new_d[4] = P_new[(int32_T)p[10] - 1];
      P_new_e[0] = P_new[(int32_T)p[6] + 10];
      P_new_e[1] = P_new[(int32_T)p[7] + 10];
      P_new_e[2] = P_new[(int32_T)p[8] + 10];
      P_new_e[3] = P_new[(int32_T)p[9] + 10];
      P_new_e[4] = P_new[(int32_T)p[10] + 10];
      for (i = 0; i < 11; i++) {
        P_LPs[i] = (*(real32_T (*)[11])&P_new[0])[i];
      }

      LX2_interp1_o5(P_new_d, P_new_e, P_LPs, *(real32_T (*)[11])&P_new[11], inst);
    } else if (LX2_sum(P_LPs, inst) == 6.0F) {
      P_new_b[0] = P_new[(int32_T)p[5] - 1];
      P_new_b[1] = P_new[(int32_T)p[6] - 1];
      P_new_b[2] = P_new[(int32_T)p[7] - 1];
      P_new_b[3] = P_new[(int32_T)p[8] - 1];
      P_new_b[4] = P_new[(int32_T)p[9] - 1];
      P_new_b[5] = P_new[(int32_T)p[10] - 1];
      P_new_c[0] = P_new[(int32_T)p[5] + 10];
      P_new_c[1] = P_new[(int32_T)p[6] + 10];
      P_new_c[2] = P_new[(int32_T)p[7] + 10];
      P_new_c[3] = P_new[(int32_T)p[8] + 10];
      P_new_c[4] = P_new[(int32_T)p[9] + 10];
      P_new_c[5] = P_new[(int32_T)p[10] + 10];
      for (i = 0; i < 11; i++) {
        P_LPs[i] = (*(real32_T (*)[11])&P_new[0])[i];
      }

      LX2_interp1_o5p(P_new_b, P_new_c, P_LPs, *(real32_T (*)[11])&P_new[11], inst);
    } else if (LX2_sum(P_LPs, inst) == 7.0F) {
      P_new_9[0] = P_new[(int32_T)p[4] - 1];
      P_new_9[1] = P_new[(int32_T)p[5] - 1];
      P_new_9[2] = P_new[(int32_T)p[6] - 1];
      P_new_9[3] = P_new[(int32_T)p[7] - 1];
      P_new_9[4] = P_new[(int32_T)p[8] - 1];
      P_new_9[5] = P_new[(int32_T)p[9] - 1];
      P_new_9[6] = P_new[(int32_T)p[10] - 1];
      P_new_a[0] = P_new[(int32_T)p[4] + 10];
      P_new_a[1] = P_new[(int32_T)p[5] + 10];
      P_new_a[2] = P_new[(int32_T)p[6] + 10];
      P_new_a[3] = P_new[(int32_T)p[7] + 10];
      P_new_a[4] = P_new[(int32_T)p[8] + 10];
      P_new_a[5] = P_new[(int32_T)p[9] + 10];
      P_new_a[6] = P_new[(int32_T)p[10] + 10];
      for (i = 0; i < 11; i++) {
        P_LPs[i] = (*(real32_T (*)[11])&P_new[0])[i];
      }

      LX2_interp1_o5pn(P_new_9, P_new_a, P_LPs, *(real32_T (*)[11])&P_new[11], inst);
    } else if (LX2_sum(P_LPs, inst) == 8.0F) {
      P_new_7[0] = P_new[(int32_T)p[3] - 1];
      P_new_7[1] = P_new[(int32_T)p[4] - 1];
      P_new_7[2] = P_new[(int32_T)p[5] - 1];
      P_new_7[3] = P_new[(int32_T)p[6] - 1];
      P_new_7[4] = P_new[(int32_T)p[7] - 1];
      P_new_7[5] = P_new[(int32_T)p[8] - 1];
      P_new_7[6] = P_new[(int32_T)p[9] - 1];
      P_new_7[7] = P_new[(int32_T)p[10] - 1];
      P_new_8[0] = P_new[(int32_T)p[3] + 10];
      P_new_8[1] = P_new[(int32_T)p[4] + 10];
      P_new_8[2] = P_new[(int32_T)p[5] + 10];
      P_new_8[3] = P_new[(int32_T)p[6] + 10];
      P_new_8[4] = P_new[(int32_T)p[7] + 10];
      P_new_8[5] = P_new[(int32_T)p[8] + 10];
      P_new_8[6] = P_new[(int32_T)p[9] + 10];
      P_new_8[7] = P_new[(int32_T)p[10] + 10];
      for (i = 0; i < 11; i++) {
        P_LPs[i] = (*(real32_T (*)[11])&P_new[0])[i];
      }

      LX2_interp1_o5pn4(P_new_7, P_new_8, P_LPs, *(real32_T (*)[11])&P_new[11], inst);
    } else if (LX2_sum(P_LPs, inst) == 9.0F) {
      P_new_5[0] = P_new[(int32_T)p[2] - 1];
      P_new_5[1] = P_new[(int32_T)p[3] - 1];
      P_new_5[2] = P_new[(int32_T)p[4] - 1];
      P_new_5[3] = P_new[(int32_T)p[5] - 1];
      P_new_5[4] = P_new[(int32_T)p[6] - 1];
      P_new_5[5] = P_new[(int32_T)p[7] - 1];
      P_new_5[6] = P_new[(int32_T)p[8] - 1];
      P_new_5[7] = P_new[(int32_T)p[9] - 1];
      P_new_5[8] = P_new[(int32_T)p[10] - 1];
      P_new_6[0] = P_new[(int32_T)p[2] + 10];
      P_new_6[1] = P_new[(int32_T)p[3] + 10];
      P_new_6[2] = P_new[(int32_T)p[4] + 10];
      P_new_6[3] = P_new[(int32_T)p[5] + 10];
      P_new_6[4] = P_new[(int32_T)p[6] + 10];
      P_new_6[5] = P_new[(int32_T)p[7] + 10];
      P_new_6[6] = P_new[(int32_T)p[8] + 10];
      P_new_6[7] = P_new[(int32_T)p[9] + 10];
      P_new_6[8] = P_new[(int32_T)p[10] + 10];
      for (i = 0; i < 11; i++) {
        P_LPs[i] = (*(real32_T (*)[11])&P_new[0])[i];
      }

      LX2_interp1_o5pn4l(P_new_5, P_new_6, P_LPs, *(real32_T (*)[11])&P_new[11], inst);
    } else if (LX2_sum(P_LPs, inst) == 10.0F) {
      P_new_3[0] = P_new[(int32_T)p[1] - 1];
      P_new_3[1] = P_new[(int32_T)p[2] - 1];
      P_new_3[2] = P_new[(int32_T)p[3] - 1];
      P_new_3[3] = P_new[(int32_T)p[4] - 1];
      P_new_3[4] = P_new[(int32_T)p[5] - 1];
      P_new_3[5] = P_new[(int32_T)p[6] - 1];
      P_new_3[6] = P_new[(int32_T)p[7] - 1];
      P_new_3[7] = P_new[(int32_T)p[8] - 1];
      P_new_3[8] = P_new[(int32_T)p[9] - 1];
      P_new_3[9] = P_new[(int32_T)p[10] - 1];
      P_new_4[0] = P_new[(int32_T)p[1] + 10];
      P_new_4[1] = P_new[(int32_T)p[2] + 10];
      P_new_4[2] = P_new[(int32_T)p[3] + 10];
      P_new_4[3] = P_new[(int32_T)p[4] + 10];
      P_new_4[4] = P_new[(int32_T)p[5] + 10];
      P_new_4[5] = P_new[(int32_T)p[6] + 10];
      P_new_4[6] = P_new[(int32_T)p[7] + 10];
      P_new_4[7] = P_new[(int32_T)p[8] + 10];
      P_new_4[8] = P_new[(int32_T)p[9] + 10];
      P_new_4[9] = P_new[(int32_T)p[10] + 10];
      for (i = 0; i < 11; i++) {
        P_LPs[i] = (*(real32_T (*)[11])&P_new[0])[i];
      }

      LX2_interp1_o5pn4ly(P_new_3, P_new_4, P_LPs, *(real32_T (*)[11])&P_new[11], inst);
    } else {
      if (LX2_sum(P_LPs, inst) == 11.0F) {
        for (i = 0; i < 11; i++) {
          P_LPs[i] = (*(real32_T (*)[11])&P_new[0])[i];
        }

        for (i = 0; i < 11; i++) {
          P_new_1[i] = (*(real32_T (*)[11])&P_new[11])[i];
        }

        for (i = 0; i < 11; i++) {
          P_new_2[i] = (*(real32_T (*)[11])&P_new[0])[i];
        }

        LX2_interp1_o5pn4ly1(P_LPs, P_new_1, P_new_2, *(real32_T (*)[11])&P_new
                             [11], inst);
      }
    }

    /*  write new interpolated values to Output */
    for (i = 0; i < 11; i++) {
      localB->OUT_offset[i] = P_new[11 + i];
      localB->OUT_measured[i] = (P_new[22 + i] != 0.0F);
    }

    /* % error calculation */
    /*  error between new delta_p2s value and interpolated BPOC-value -> for debugging reasons only */
    if ((aa_0 != 0.0F) && (aa_0 != 11.0F)) {
      tmp_0[0] = (real32_T)((int32_T)aa - 1) * 10.0F;
      tmp_0[1] = (real32_T)((int32_T)(aa + 1.0F) - 1) * 10.0F;
      P_new_0[0] = P_new[(int32_T)aa + 10];
      P_new_0[1] = P_new[(int32_T)(aa + 1.0F) + 10];
      slope = y - LX2_interp1_o5pn4ly1e(tmp_0, P_new_0, x, inst);
    } else {
      /*  a2==single(11) */
      slope = y - P_new[(int32_T)aa_0 + 10];
    }

    localB->DBUG_a[0] = aa;
    localB->DBUG_a[1] = aa_0;

    /*  a1, a2 ... results of my_detect */
    localB->DBUG_b[0] = b;
    localB->DBUG_b[1] = b_0;

    /*  b1, b2 ... results of my_split */
    tmp[0] = 0.0F;
    tmp[1] = Lp_idx_0 - 1.0F;
    tmp[2] = 10.0F;
    tmp[3] = Lp_idx - 1.0F;
    LX2_rdivide(tmp, 10.0, localB->DBUG_Lp, inst);

    /*  Lp ... location of leanox points on map (indices). Set DBUG_Lp(4,1) to -1 if Lp_c not enabled */
    localB->DBUG_s[0] = DBUG_sInt;
    localB->DBUG_s[1] = DBUG_sExt_left;
    localB->DBUG_s[2] = DBUG_sExt_right;

    /*  DBUG_sInt ... slope between affected nodes, DBUG_sExt_left ... extrapolation slope to the left side, DBUG_sExt_right ... extrapolation slope to the left side */
  } else {
    /*  if function is disabled... Input == Output */
    for (i = 0; i < 11; i++) {
      localB->OUT_offset[i] = rtu_IN_offset[i];
      localB->OUT_measured[i] = rtu_IN_measured[i];
    }

    slope = 0.0F;

    /*  set error to zero -> for debugging reasons only */
    localB->DBUG_a[0] = -1.0F;
    localB->DBUG_a[1] = -1.0F;

    /*  a1, a2 ... results of my_detect | % set var to -1 -> for debugging reasons only */
    localB->DBUG_b[0] = -1.0F;
    localB->DBUG_b[1] = -1.0F;

    /*  b1, b2 ... results of my_split | % set var to -1 -> for debugging reasons only */
    localB->DBUG_Lp[0] = -1.0F;
    localB->DBUG_Lp[1] = -1.0F;
    localB->DBUG_Lp[2] = -1.0F;
    localB->DBUG_Lp[3] = -1.0F;

    /*  Lp ... location of leanox points on map (indices) | % set var to -1 -> for debugging reasons only */
    localB->DBUG_s[0] = -1.0F;
    localB->DBUG_s[1] = -1.0F;
    localB->DBUG_s[2] = -1.0F;

    /*  s ... calculated slopes (Interpolation/Extrapolation)  | % set var to -1 -> for debugging reasons only */
  }

  /* '<S15>:1:3' */
  localB->e = slope;
}

/*
 * Output and update for atomic system:
 *    '<S37>/TON'
 *    '<S54>/TON'
 */
void LX2_TON(boolean_T rtu_IN, real32_T rtu_PT, rtB_TON_LX2 *localB,
             rtDW_TON_LX2 *localDW, struct fLX2* inst)
{
  /* local block i/o variables */
  boolean_T rtb_LogicalOperator2_g;
  boolean_T rtb_RelationalOperator_o;

  /* Logic: '<S47>/Logical Operator2' */
  rtb_LogicalOperator2_g = !rtu_IN;

  /* DiscreteIntegrator: '<S47>/Discrete-Time Integrator' */
  if (rtb_LogicalOperator2_g || (localDW->DiscreteTimeIntegrator_PrevRese != 0))
  {
    localDW->DiscreteTimeIntegrator_DSTATE = 0.0F;
  }

  localB->DiscreteTimeIntegrator = localDW->DiscreteTimeIntegrator_DSTATE;

  /* End of DiscreteIntegrator: '<S47>/Discrete-Time Integrator' */

  /* RelationalOperator: '<S47>/Relational Operator' */
  rtb_RelationalOperator_o = (localB->DiscreteTimeIntegrator >= rtu_PT);

  /* Logic: '<S47>/Logical Operator3' */
  localB->LogicalOperator3 = (rtb_RelationalOperator_o && rtu_IN);

  /* Update for DiscreteIntegrator: '<S47>/Discrete-Time Integrator' incorporates:
   *  DataTypeConversion: '<S48>/Conversion'
   *  Logic: '<S47>/Logical Operator'
   *  Logic: '<S47>/Logical Operator1'
   */
  localDW->DiscreteTimeIntegrator_DSTATE += (real32_T)
    ((!rtb_RelationalOperator_o) && rtu_IN) * 0.1F;
  if (rtb_LogicalOperator2_g) {
    localDW->DiscreteTimeIntegrator_PrevRese = 1;
  } else {
    localDW->DiscreteTimeIntegrator_PrevRese = 0;
  }

  /* End of Update for DiscreteIntegrator: '<S47>/Discrete-Time Integrator' */
}

/*
 * Initial conditions for atomic system:
 *    '<S8>/Filter1'
 *    '<S51>/Filter'
 *    '<S51>/Filter1'
 */
void LX2_Filter1_Init(rtDW_Filter1_LX2 *localDW, struct fLX2* inst)
{
  /* InitializeConditions for DiscreteIntegrator: '<S50>/Discrete-Time Integrator' */
  localDW->DiscreteTimeIntegrator_IC_LOADI = 1U;
}

/*
 * Output and update for atomic system:
 *    '<S8>/Filter1'
 *    '<S51>/Filter'
 *    '<S51>/Filter1'
 */
void LX2_Filter1(uint16_T rtu_T_filt, boolean_T rtu_reset, real32_T rtu_x0,
                 rtB_Filter1_LX2 *localB, rtDW_Filter1_LX2 *localDW, struct fLX2* inst)
{
  /* local block i/o variables */
  boolean_T rtb_LogicalOperator_j;
  boolean_T rtb_RelationalOperator_ly;
  real32_T tmp;

  /* RelationalOperator: '<S50>/Relational Operator' incorporates:
   *  Constant: '<S50>/Constant'
   *  DataTypeConversion: '<S50>/Data Type Conversion2'
   */
  rtb_RelationalOperator_ly = (rtu_T_filt > 0);

  /* Logic: '<S50>/Logical Operator' incorporates:
   *  Logic: '<S50>/Logical Operator1'
   */
  rtb_LogicalOperator_j = (rtu_reset || (!rtb_RelationalOperator_ly));

  /* DiscreteIntegrator: '<S50>/Discrete-Time Integrator' */
  if (localDW->DiscreteTimeIntegrator_IC_LOADI != 0) {
    localDW->DiscreteTimeIntegrator_DSTATE = rtu_x0;
  }

  if (rtb_LogicalOperator_j || (localDW->DiscreteTimeIntegrator_PrevRese != 0))
  {
    localDW->DiscreteTimeIntegrator_DSTATE = rtu_x0;
  }

  /* Switch: '<S50>/Switch' incorporates:
   *  DiscreteIntegrator: '<S50>/Discrete-Time Integrator'
   */
  if (rtb_RelationalOperator_ly) {
    localB->Switch = localDW->DiscreteTimeIntegrator_DSTATE;
  } else {
    localB->Switch = rtu_x0;
  }

  /* End of Switch: '<S50>/Switch' */

  /* Update for DiscreteIntegrator: '<S50>/Discrete-Time Integrator' */
  localDW->DiscreteTimeIntegrator_IC_LOADI = 0U;

  /* Switch: '<S55>/Switch' incorporates:
   *  Constant: '<S55>/Constant2'
   *  DataTypeConversion: '<S50>/Data Type Conversion2'
   *  RelationalOperator: '<S55>/Relational Operator'
   */
  if (0.1F >= (real32_T)rtu_T_filt) {
    tmp = 0.1F;
  } else {
    tmp = (real32_T)rtu_T_filt;
  }

  /* End of Switch: '<S55>/Switch' */

  /* Update for DiscreteIntegrator: '<S50>/Discrete-Time Integrator' incorporates:
   *  DiscreteIntegrator: '<S50>/Discrete-Time Integrator'
   *  Product: '<S50>/Divide4'
   *  Sum: '<S50>/Sum4'
   */
  localDW->DiscreteTimeIntegrator_DSTATE += (rtu_x0 -
    localDW->DiscreteTimeIntegrator_DSTATE) / tmp * 0.1F;
  if (rtb_LogicalOperator_j) {
    localDW->DiscreteTimeIntegrator_PrevRese = 1;
  } else {
    localDW->DiscreteTimeIntegrator_PrevRese = 0;
  }
}

/* Function for MATLAB Function: '<S8>/MATLAB Function' */
static void LX2_my_BPOC_enable_h(const real32_T splitfactor[4], boolean_T
  bLX2_enable, const real32_T rThreshold_save2map[2], boolean_T
  bExt_BPOC_learning_Stop, boolean_T bBPOC_enable[4], boolean_T
  bSave_BPOC_enable[4], struct fLX2* inst)
{
  /* % my_BPOC_enable */
  bSave_BPOC_enable[0] = (bLX2_enable && (splitfactor[0] > rThreshold_save2map[0])
    && (splitfactor[2] < 1.0F - rThreshold_save2map[1]) &&
    (!bExt_BPOC_learning_Stop));
  bBPOC_enable[0] = (splitfactor[0] > 0.0F);
  bSave_BPOC_enable[1] = (bLX2_enable && (splitfactor[1] > rThreshold_save2map[0])
    && (splitfactor[2] < 1.0F - rThreshold_save2map[1]) &&
    (!bExt_BPOC_learning_Stop));
  bBPOC_enable[1] = (splitfactor[1] > 0.0F);
  bSave_BPOC_enable[2] = (bLX2_enable && (splitfactor[2] > rThreshold_save2map[1])
    && (!bExt_BPOC_learning_Stop));
  bBPOC_enable[2] = (splitfactor[2] > 0.0F);
  bSave_BPOC_enable[3] = (bLX2_enable && (splitfactor[3] > rThreshold_save2map[1])
    && (!bExt_BPOC_learning_Stop));
  bBPOC_enable[3] = (splitfactor[3] > 0.0F);
}

/* Function for MATLAB Function: '<S8>/MATLAB Function' */
static void LX2_my_BPOC_enable(const real32_T splitfactor[4], boolean_T
  bLX2_enable, const real32_T rThreshold_save2map[2], boolean_T
  bExt_BPOC_learning_Stop, boolean_T bBPOC_enable[4], boolean_T
  bSave_BPOC_enable[4], struct fLX2* inst)
{
  /* % my_BPOC_enable */
  bSave_BPOC_enable[0] = (bLX2_enable && (splitfactor[0] > rThreshold_save2map[0])
    && (splitfactor[2] < 1.0F - rThreshold_save2map[1]) &&
    (!bExt_BPOC_learning_Stop));
  bBPOC_enable[0] = (splitfactor[0] > 0.0F);
  bSave_BPOC_enable[1] = (bLX2_enable && (splitfactor[1] > rThreshold_save2map[0])
    && (splitfactor[2] < 1.0F - rThreshold_save2map[1]) &&
    (!bExt_BPOC_learning_Stop));
  bBPOC_enable[1] = (splitfactor[1] > 0.0F);
  bSave_BPOC_enable[2] = (bLX2_enable && (splitfactor[2] > rThreshold_save2map[1])
    && (!bExt_BPOC_learning_Stop));
  bBPOC_enable[2] = (splitfactor[2] > 0.0F);
  bSave_BPOC_enable[3] = (bLX2_enable && (splitfactor[3] > rThreshold_save2map[1])
    && (!bExt_BPOC_learning_Stop));
  bBPOC_enable[3] = (splitfactor[3] > 0.0F);
}

/* Function for MATLAB Function: '<S8>/MATLAB Function' */
static void LX2_my_gasmixing(uint16_T iIdx_Gtyp_Dem, real32_T rGT_QualMix_1_2,
  real32_T rGT_RatioMix, boolean_T bLX2_enable, const real32_T
  rThreshold_save2map[2], boolean_T bExt_BPOC_learning_Stop, real32_T
  splitfactor_Gas[4], boolean_T bBPOC_enable[4], boolean_T bSave_BPOC_enable[4], struct fLX2* inst)
{
  real32_T tmp[2];

  /*  function undesired_operating */
  /* % function my_gasmixing <<LX2_FunReq-26>> */
  /*  define output vectors */
  if (iIdx_Gtyp_Dem < 4) {
    splitfactor_Gas[0] = (1.0F - rGT_QualMix_1_2) * (1.0F - rGT_RatioMix);
    splitfactor_Gas[1] = (1.0F - rGT_RatioMix) * rGT_QualMix_1_2;
    splitfactor_Gas[2] = rGT_RatioMix;
    splitfactor_Gas[3] = 0.0F;
    LX2_my_BPOC_enable(splitfactor_Gas, bLX2_enable, rThreshold_save2map,
                       bExt_BPOC_learning_Stop, bBPOC_enable, bSave_BPOC_enable, inst);
  } else if (iIdx_Gtyp_Dem == 4) {
    splitfactor_Gas[0] = 0.0F;
    splitfactor_Gas[1] = 0.0F;
    splitfactor_Gas[2] = 0.0F;
    splitfactor_Gas[3] = 1.0F;
    tmp[0] = 0.0F;
    tmp[1] = 0.0F;
    LX2_my_BPOC_enable_h(splitfactor_Gas, bLX2_enable, tmp,
                         bExt_BPOC_learning_Stop, bBPOC_enable,
                         bSave_BPOC_enable, inst);
  } else {
    /*  undefined Gastype */
    splitfactor_Gas[0] = 0.0F;
    splitfactor_Gas[1] = 0.0F;
    splitfactor_Gas[2] = 0.0F;
    splitfactor_Gas[3] = 0.0F;
    tmp[0] = 1.0F;
    tmp[1] = 1.0F;
    LX2_my_BPOC_enable_h(splitfactor_Gas, bLX2_enable, tmp,
                         bExt_BPOC_learning_Stop, bBPOC_enable,
                         bSave_BPOC_enable, inst);
  }
}

/* Model step function */
void LX2_step(struct fLX2* inst)
{
  /* local block i/o variables */
  real32_T rtb_rLX2_inLimitSetup_Time;
  real32_T rtb_rPr_Leanox_Dev;
  real32_T rtb_rP_Set_Norm;
  real32_T rtb_DataTypeConversion;
  real32_T rtb_Gain7;
  real32_T rtb_Delay2[11];
  real32_T rtb_Sum1;
  real32_T rtb_Lp2Lp3Lp_c[3];
  real32_T rtb_mbar2bar2;
  real32_T rtb_mbar2bar3;
  real32_T rtb_mbar2bar4;
  real32_T rtb_Switch1[11];
  real32_T rtb_Delay2_e[11];
  real32_T rtb_Sum1_e;
  real32_T rtb_Lp2Lp3Lp_c_n[3];
  real32_T rtb_mbar2bar2_e;
  real32_T rtb_mbar2bar3_h;
  real32_T rtb_mbar2bar4_m;
  real32_T rtb_Switch1_m[11];
  real32_T rtb_Delay2_o[11];
  real32_T rtb_Sum1_b;
  real32_T rtb_Lp2Lp3Lp_c_l[3];
  real32_T rtb_mbar2bar2_o;
  real32_T rtb_mbar2bar3_o;
  real32_T rtb_mbar2bar4_e;
  real32_T rtb_Switch1_i[11];
  real32_T rtb_Delay2_o1[11];
  real32_T rtb_Sum1_h;
  real32_T rtb_Lp2Lp3Lp_c_e[3];
  real32_T rtb_mbar2bar2_m;
  real32_T rtb_mbar2bar3_a;
  real32_T rtb_mbar2bar4_g;
  real32_T rtb_Switch1_it[11];
  real32_T rtb_InterpolateBPOCatLp_c25load;
  real32_T rtb_InterpolateBPOC;
  real32_T rtb_InterpolateBPOCatLp_c25lo_h;
  real32_T rtb_InterpolateBPOC_k;
  real32_T rtb_InterpolateBPOCatLp_c25lo_l;
  real32_T rtb_InterpolateBPOC_h;
  real32_T rtb_InterpolateBPOCatLp_c25lo_e;
  real32_T rtb_InterpolateBPOC_a;
  real32_T rtb_Selector12;
  real32_T rtb_Switch2_b;
  real32_T rtb_Abs;
  real32_T rtb_Divide;
  real32_T rtb_Switch2_l;
  uint16_T rtb_iFiltConst_LeanoxDev_Steady;
  uint16_T rtb_iFiltConst_P_set_SteadyStat;
  uint16_T rtb_iFilterConst_P_set;
  uint16_T rtb_iWeight_Lp_0kW;
  uint16_T rtb_iWeight_Lp_b;
  uint16_T rtb_iWeight_Lp_a;
  uint16_T rtb_iWeight_Lp_c;
  uint16_T rtb_iWeight_Lp_0kW_e;
  uint16_T rtb_iWeight_Lp_b_c;
  uint16_T rtb_iWeight_Lp_a_m;
  uint16_T rtb_iWeight_Lp_c_m;
  uint16_T rtb_iWeight_Lp_0kW_d;
  uint16_T rtb_iWeight_Lp_b_a;
  uint16_T rtb_iWeight_Lp_a_j;
  uint16_T rtb_iWeight_Lp_c_f;
  uint16_T rtb_iWeight_Lp_0kW_k;
  uint16_T rtb_iWeight_Lp_b_e;
  uint16_T rtb_iWeight_Lp_a_h;
  uint16_T rtb_iWeight_Lp_c_e;
  boolean_T rtb_LogicalOperator1;
  boolean_T rtb_LogicalOperator3;
  boolean_T rtb_LogicalOperator4_n;
  boolean_T rtb_LogicalOperator8_g;
  boolean_T rtb_LogicalOperator7_m;
  boolean_T rtb_bLp_c_ena;
  boolean_T rtb_Delay1[11];
  boolean_T rtb_LogicalOperator7_e;
  boolean_T rtb_bLp_c_ena_i;
  boolean_T rtb_Delay1_g[11];
  boolean_T rtb_LogicalOperator7_l;
  boolean_T rtb_bLp_c_ena_h;
  boolean_T rtb_Delay1_l[11];
  boolean_T rtb_LogicalOperator7_i;
  boolean_T rtb_bLp_c_ena_n;
  boolean_T rtb_Delay1_c[11];
  boolean_T rtb_LogicalOperator4_g;
  boolean_T rtb_LogicalOperator2_de;
  boolean_T rtb_Reset;
  boolean_T rtb_LogicalOperator_d;
  boolean_T didZcEventOccur;
  boolean_T bCtrl_enable;
  boolean_T bCtrl_freeze;
  boolean_T bEng_misfire;
  boolean_T b_bEng_knock;
  real32_T b_y;
  real32_T rtb_Switch2_kt;
  real32_T rtb_Switch7;
  real32_T rtb_Gain3;
  boolean_T rtb_u;
  boolean_T rtb_u_b;
  boolean_T rtb_LogicalOperator2;
  boolean_T rtb_LogicalOperator3_e;
  real32_T rtb_Switch_nq;
  boolean_T rtb_Compare_n;
  real32_T rtb_rNOx_act_g;
  boolean_T rtb_LogicalOperator6_a;
  boolean_T rtb_LogicalOperator_f;
  boolean_T rtb_bSave_BPOC_enable[4];
  real32_T rtb_rP_Lp_c[5];
  real32_T rtb_rPr_LX2_offset_Lp_c[5];
  real32_T rtb_rPr_LX2_offset_Lp_a[5];
  real32_T rtb_rPr_LX2_offset_Lp_b[5];
  boolean_T rtb_LogicalOperator5_k;
  real32_T rtb_splitfactor_Gas[4];
  real32_T rtb_Switch3;
  real32_T rtb_LowerLimit_factor;
  boolean_T rtb_bBPOC_enable_a[4];
  real32_T rtb_SumofElements2;
  real32_T rtb_SumofElements1;
  real32_T rtb_SumofElements_o;
  real32_T rtb_SumofElements;
  real32_T rtb_DiscreteTimeIntegrator;
  real32_T rtb_Sum2_e;
  boolean_T rtb_bLX2_save[5];
  real32_T rtb_Product4[11];
  real32_T rtb_Product5[11];
  real32_T rtb_Product6[11];
  real32_T rtb_Product7[11];
  int8_T rtb_Switch5_kl[11];
  int8_T rtb_Switch4[11];
  int8_T rtb_Switch6_j[11];
  int8_T rtb_rLX2_BPOC[11];
  real32_T rtb_Switch2[11];
  real32_T rtb_Switch2_j[11];
  real32_T rtb_Switch2_k[11];
  real32_T rtb_Switch2_kq[11];
  real32_T rtb_Switch6;
  real32_T rtb_UnitDelay3;
  boolean_T rtb_RelationalOperator_b;
  boolean_T rtb_UnitDelay1;
  real32_T rtb_UnitDelay2;
  int32_T i;
  real32_T tmp[2];
  real32_T rtb_splitfactor_VISU_idx;
  boolean_T rtb_Switch2_a_idx;
  boolean_T rtb_Switch2_a_idx_0;
  boolean_T rtb_Switch2_a_idx_1;
  boolean_T rtb_Switch2_a_idx_2;
  uint32_T tmp_0;
  real_T rtb_Sum2_e_0;
  real32_T tmp_1;
  int32_T rtb_splitfactor_Gas_0;
  real_T tmp_2;
  int32_T rtb_splitfactor_Gas_1;
  int32_T rtb_splitfactor_Gas_2;
  int32_T rtb_splitfactor_Gas_3;

  /* S-Function (bur_bus_in): '<Root>/Bus Input' */
  LX2_B.BusInput = inst->IN;

  /* Switch: '<S7>/Switch3' incorporates:
   *  Constant: '<S7>/Constant1'
   */
  if (LX2_B.BusInput.bLX2_fastRamp) {
    rtb_Switch7 = LX2_B.BusInput.rLX2_fastRampMult;
  } else {
    rtb_Switch7 = 1.0F;
  }
```
